(* IEC 61131-3 sources: elnaProjects/ElpcLogic/PomarKc7Changed/build_USO_ecl, 1 file *)

(* ---- plc.st ---- *)
TYPE
  TYPE_PhaseAlgoritmAction : (_run, _reset);
  TYPE_DualStateImAction : (_on, _off);
  struct_SectionSwitch : STRUCT
    inCommand : WORD;
    status : DWORD;
    onStatus : BYTE;
    inOpcCommandsDisabled : BOOL;
    sdvig : BOOL;
    Ns : BOOL;
    CommandFault : BOOL;
    Accident : BOOL;
    Local : BOOL;
    Distance : BOOL;
    OpcCommandsDisabled : BOOL;
    lastCmdIsOn : BOOL;
    offKNA : BOOL;
    basketStatus : BYTE;
    ISVALIDREF_statOn : BOOL;
    ISVALIDREF_statOff : BOOL;
    ISVALIDREF_cmdOn : BOOL;
    ISVALIDREF_cmdOff : BOOL;
    ISVALIDREF_inBreakCmdOn : BOOL;
    ISVALIDREF_inBreakCmdOff : BOOL;
    BreakCmdOn : BOOL;
    BreakCmdOff : BOOL;
    ISVALIDREF_basketRolledIn : BOOL;
    ISVALIDREF_basketRolledOut : BOOL;
    ISVALIDREF_basketTest : BOOL;
    inCommand_Alg : WORD;
    inCommand_ARM : WORD;
    cmdOn : BOOL;
    cmdOff : BOOL;
    reliability : BOOL;
  END_STRUCT;
  struct_ReserveIM2 : STRUCT
    var1 : BOOL;
    var2 : BOOL;
  END_STRUCT;
  struct_DiProtection : STRUCT
    delay : TIME;
    inTag : BYTE;
    inRunOnStart : BOOL;
    inCanRun : BOOL;
    inOpcCommandsDisabled : BOOL;
    inCommand : WORD;
    inCommand_Alg : WORD;
    inCommand_ARM : WORD;
    Tag : BYTE;
    status : DWORD;
    CanRun : BOOL;
    OpcCommandsDisabled : BOOL;
    isRunning : BOOL;
    HasError : BOOL;
    isEnded : BOOL;
    Remont : BOOL;
    Check : BOOL;
    Signaling : BOOL;
    SignalingTP : BOOL;
    RunOnStart : BOOL;
  END_STRUCT;
  TYPE_ReliableBit : STRUCT
    value : BOOL;
    reliability : BOOL;
    _inversed : BOOL;
  END_STRUCT;
  struct_DI : STRUCT
    imit : BOOL;
    value : WORD;
    reliability : WORD;
    bits : ARRAY [0..15] OF TYPE_ReliableBit;
    blConnect : BOOL;
  END_STRUCT;
  struct_AiProtection : STRUCT
    controlLimit : BYTE;
    delay : TIME;
    inTag : BYTE;
    inRunOnStart : BOOL;
    inCanRun : BOOL;
    inOpcCommandsDisabled : BOOL;
    inCommand : WORD;
    inCommand_Alg : WORD;
    inCommand_ARM : WORD;
    Tag : BYTE;
    status : DWORD;
    CanRun : BOOL;
    OpcCommandsDisabled : BOOL;
    isRunning : BOOL;
    HasError : BOOL;
    isEnded : BOOL;
    Remont : BOOL;
    Check : BOOL;
    Signaling : BOOL;
    SignalingTP : BOOL;
    RunOnStart : BOOL;
  END_STRUCT;
  ProtectionsConfig : STRUCT
    Topornogo_podshipnika_EDT_1 : struct_AiProtection;
    Toy_podshipnika_EDT_2 : struct_AiProtection;
    Toy_podshipnika_kol_EDT_3 : struct_AiProtection;
    Toy_podshipnika_kol_EDT_4 : struct_AiProtection;
    To_podshipnika_shest_red_EDT_5 : struct_AiProtection;
    To_podshipnika_shest_red_EDT_6 : struct_AiProtection;
    To_podshipnika_N_EDT_7 : struct_AiProtection;
    To_podshipnika_svob_konca_EDT_8 : struct_AiProtection;
    Ty_podshipnika_rab_kol_EDT_9 : struct_AiProtection;
    Typornogo_podshipnika_nerab_kolodok_HT_10 : struct_AiProtection;
    Tgaza_na_vyhode_H : struct_AiProtection;
    Os_sdvig_nagnetatelja_plus : struct_AiProtection;
    Os_sdvig_nagnetatelja_minus : struct_AiProtection;
    Pgaza_na_vyhode_nagnetatelia_GPA_STOP : struct_AiProtection;
    Pgaza_na_vhode_nagnetatelia_GPA_STOP : struct_AiProtection;
    Pgaza_na_vyhode_nagnetatelia : struct_AiProtection;
    dPmaslo_gaz : struct_AiProtection;
    Pmaslo_sm_nizkoe : struct_AiProtection;
    Pmaslo_sm_vysokoe : struct_AiProtection;
    Vibro_skorost_OPED_T1 : struct_AiProtection;
    Vibro_skorost_OPED_T2 : struct_AiProtection;
    Vibro_skorost_OYP_kolesa_ED_T3 : struct_AiProtection;
    Vibro_skorost_OP_kolesa_RH_T4 : struct_AiProtection;
    Vibro_skorost_OP_shesterni_RED_T5 : struct_AiProtection;
    Vibro_skorost_OP_shesterni_RED_T6 : struct_AiProtection;
    dPmaslo_gaz_less100 : struct_DiProtection;
    Reg_vozb_off : struct_DiProtection;
    Fail_chastotnii_pusk : struct_DiProtection;
    Off_avar_vikluchatel : struct_DiProtection;
    AOKC_SHKC : struct_DiProtection;
    AO_PRU : struct_DiProtection;
    AO_ot_SHU : struct_DiProtection;
    mvOff : struct_DiProtection;
    Kran1_sdvig : struct_DiProtection;
    Kran2_sdvig : struct_DiProtection;
  END_STRUCT;
  struct_singleSignal : STRUCT
    reliability : BOOL;
    inverse : BOOL;
    DelayOn : TIME;
    DelayOff : TIME;
    Q : BOOL;
    status : DWORD;
    Disabled_Sig : BOOL;
  END_STRUCT;
  IM_singleSignals : STRUCT
    dP_maslo_gaz_Less100 : struct_singleSignal;
    dp_kran1_Less100 : struct_singleSignal;
    Razreshenie_zagruzki_dvig : struct_singleSignal;
    Vozbud_gotovnost : struct_singleSignal;
    Vozbud_neispr_tsepey_upr_AVR_pit : struct_singleSignal;
    Vozbud_neispravnost : struct_singleSignal;
    SHAVR1_v_rabote : struct_singleSignal;
    SHAVR2_v_rabote : struct_singleSignal;
    Avariinoe_otkluch_vikluchatelya : struct_singleSignal;
    Assinhronnii_hod_peregruzka : struct_singleSignal;
    SHU_v_GPA_vkluch : struct_singleSignal;
    SHP_v_GPA_vkluch : struct_singleSignal;
    QF1_on : struct_singleSignal;
    QF2_on : struct_singleSignal;
    QF23_on : struct_singleSignal;
    QF4_QF5_on : struct_singleSignal;
    QF6_QF7_on : struct_singleSignal;
    QF8_QF9_on : struct_singleSignal;
    QF10_QF11_on : struct_singleSignal;
    QF12_QF13_on : struct_singleSignal;
    QF14_QF15_on : struct_singleSignal;
    QF22_on : struct_singleSignal;
    NS_G1_G2 : struct_singleSignal;
    NS_G3_G4 : struct_singleSignal;
    NS_G15_G16 : struct_singleSignal;
    NS_G17 : struct_singleSignal;
    NS_G5_G6 : struct_singleSignal;
    NS_G7_G8 : struct_singleSignal;
    NS_G18_G19 : struct_singleSignal;
    NS_G10_G11 : struct_singleSignal;
    NS_G13_G14 : struct_singleSignal;
    Uroven_masla_akkum : struct_singleSignal;
    NKU1_GPA_on : struct_singleSignal;
    NKU2_GPA_on : struct_singleSignal;
    AO_KC_ot_SHKS : struct_singleSignal;
    AO_GPA_ot_SHU : struct_singleSignal;
    BEAO_srabotal : struct_singleSignal;
    Chastotny_pusk : struct_singleSignal;
    Neuspesh_chastotny_pusk : struct_singleSignal;
    Rezhim_ruchnogo_regulirovaniya : struct_singleSignal;
    Osnovnoy_regul_off : struct_singleSignal;
    Voltage_sekcii_norm : struct_singleSignal;
    Reactorny_pusk : struct_singleSignal;
    NO_GPA_ot_SHU : struct_singleSignal;
    AO_GPA_ot_PRU : struct_singleSignal;
    Nalichie_BP1 : struct_singleSignal;
    Nalichie_BP2 : struct_singleSignal;
    Nalichie_BP3 : struct_singleSignal;
    Nalichie_BP4 : struct_singleSignal;
    Nalichie_BP5 : struct_singleSignal;
    Nalichie_BP6 : struct_singleSignal;
    Nalichie_BP7_BP8 : struct_singleSignal;
    Nalichie_BP9_BP10 : struct_singleSignal;
    Nalichie_cepei_upravlen_mv : struct_singleSignal;
    Nalichie_220BEAO : struct_singleSignal;
    Nalichie_per_220_na_vhode : struct_singleSignal;
    Nalichie_post_220_na_vhode : struct_singleSignal;
    Nalichie_BP11 : struct_singleSignal;
    Nalichie_BP12 : struct_singleSignal;
    Dver_SHU_pered_otkrita : struct_singleSignal;
    Dver_SHU_zad_otkrita : struct_singleSignal;
    EO_GPA_ot_knopki_SHU : struct_singleSignal;
    EO_EGPA_ot_PRY : struct_singleSignal;
    Synchroniz_rezhima_K1 : struct_singleSignal;
    Potok_ms_posle_AVOM : struct_singleSignal;
  END_STRUCT;
  DiConfig : STRUCT
    di_0 : struct_DI;
    di_1 : struct_DI;
    di_2 : struct_DI;
    di_3 : struct_DI;
    di_4 : struct_DI;
    di_5 : struct_DI;
    di_6 : struct_DI;
    di_7 : struct_DI;
    di_8 : struct_DI;
    di_9 : struct_DI;
    di_10 : struct_DI;
    di_11 : struct_DI;
    di_12 : struct_DI;
    di_13 : struct_DI;
    di_14 : struct_DI;
    di_15 : struct_DI;
    di_16 : struct_DI;
    di_17 : struct_DI;
    di_18 : struct_DI;
    di_19 : struct_DI;
    di_20 : struct_DI;
    di_21 : struct_DI;
  END_STRUCT;
  struct_AO : STRUCT
    nValue : LREAL;
    blConnect : BOOL;
    outLL : LREAL;
    outHL : LREAL;
    newLL : LREAL;
    newHL : LREAL;
    newLL_ISVALIDREF : BOOL;
    newHL_ISVALIDREF : BOOL;
    inCommand : WORD;
    Value : LREAL;
    status : DWORD;
    LL : LREAL;
    HL : LREAL;
    OpcCommandsDisabled : BOOL;
  END_STRUCT;
  AOConfig : STRUCT
    Reserv_AO_1 : struct_AO;
    Reserv_AO_2 : struct_AO;
  END_STRUCT;
  struct_AI : STRUCT
    value : LREAL;
    status : DWORD;
    interval : BYTE;
    inCommand : WORD;
    blConnect : BOOL;
    dLL : LREAL;
    dHL : LREAL;
    dLA : LREAL;
    dHA : LREAL;
    dLW : LREAL;
    dHW : LREAL;
    LL : LREAL;
    HL : LREAL;
    LA : LREAL;
    HA : LREAL;
    LW : LREAL;
    HW : LREAL;
    ISVALIDREF_LA : BOOL;
    ISVALIDREF_HA : BOOL;
    ISVALIDREF_LW : BOOL;
    ISVALIDREF_HW : BOOL;
    inpLL : LREAL;
    inpHL : LREAL;
    CurrentShotCircuit : LREAL;
    CurrentBreakCircuit : LREAL;
    maxChangeSpeed : LREAL;
    maxChangeSpeedDown : LREAL;
    ChangeSpeed : LREAL;
    histeresis : LREAL;
    aperturFilter : LREAL;
    exponentialFilter : LREAL;
    rassoglasovanie : LREAL;
    OpcCommandsDisabled : BOOL;
    Disabled_LA : BOOL;
    Disabled_HA : BOOL;
    Disabled_LW : BOOL;
    Disabled_HW : BOOL;
    delayLA : TIME;
    delayLW : TIME;
    delayHW : TIME;
    delayHA : TIME;
    minValue_ISVALIDREF : BOOL;
    maxValue_ISVALIDREF : BOOL;
    minValue : LREAL;
    maxValue : LREAL;
    inOpcCommandsDisabled : BOOL;
    imit : BOOL;
    remont : BOOL;
    NS : BOOL;
    NS_Min : BOOL;
    NS_Max : BOOL;
    inCommand_Alg : WORD;
    inCommand_ARM : WORD;
    dMaxChangeSpeed : LREAL;
    dMaxChangeSpeedDown : LREAL;
  END_STRUCT;
  AiConfig : STRUCT
    Tstali_statora_kanal_1 : struct_AI;
    Tstali_statora_kanal_2 : struct_AI;
    Tstali_statora_kanal_3 : struct_AI;
    Tmedi_statora_kanal_1 : struct_AI;
    Tmedi_statora_kanal_2 : struct_AI;
    Tmedi_statora_kanal_3 : struct_AI;
    Toporno_podshipnika_EDT_1 : struct_AI;
    Toy_podshipnika_EDT_2 : struct_AI;
    Toy_podshipnika_kol_EDT_3 : struct_AI;
    Toy_podshipnika_kol_EDT_4 : struct_AI;
    Toy_podshipnika_shest_red_EDT_5 : struct_AI;
    Ty_podshipnika_red_EDT_6 : struct_AI;
    Ty_podshipnika_nagnet_EDT_7_1 : struct_AI;
    Ty_podshipnika_nagnet_EDT_7_2 : struct_AI;
    Toy_podshipnika_svobod_konca_EDT_8_1 : struct_AI;
    Toy_podshipnika_svobod_konca_EDT_8_2 : struct_AI;
    Toy_podshipnika_rab_kol_EDT_9_1 : struct_AI;
    Toy_podshipnika_rab_kol_EDT_9_2 : struct_AI;
    Toy_podshipnika_nerab_kol_EDT_10_1 : struct_AI;
    Toy_podshipnika_nerab_kol_EDT_10_2 : struct_AI;
    Tholodnogo_vozduha_ED_kanal_1 : struct_AI;
    Tholodnogo_vozduha_ED_kanal_2 : struct_AI;
    Tgorjachego_vozduha_ED_kanal_1 : struct_AI;
    Tgorjachego_vozduha_ED_kanal_2 : struct_AI;
    Tnarujnogo_vozduha : struct_AI;
    Tgaza_na_vhode_H : struct_AI;
    Tgaza_na_vyhode_H : struct_AI;
    Tmasla_do_AVOM : struct_AI;
    Tmasla_posle_AVOM : struct_AI;
    Tmasla_MB : struct_AI;
    Tmasla_MB_TEN : struct_AI;
    Tshu : struct_AI;
    Pmaslo_sm_nizkoe : struct_AI;
    Pmaslo_sm_vysokoe : struct_AI;
    Pmasla_posle_GNS : struct_AI;
    Pmasla_posle_NU : struct_AI;
    Pgaza_na_vhode_nagnetatelia : struct_AI;
    Pgaza_na_vyhode_nagnetatelia : struct_AI;
    Pimpuls_gaz : struct_AI;
    dPgaza_na_maslo_filtre : struct_AI;
    dPgaza_na_konfuzore : struct_AI;
    dPmaslo_gaz : struct_AI;
    Os_sdvig_nagnetatelja_plus : struct_AI;
    Os_sdvig_nagnetatelja_minus : struct_AI;
    Yroven_masla_MB : struct_AI;
    Kontrol_per_220V : struct_AI;
    Kontrol_post_220V : struct_AI;
    Tok_statora : struct_AI;
    Vibro_skorost_OPED_T1 : struct_AI;
    Vibro_skorost_OYPED_T2 : struct_AI;
    Vibro_skorost_OYP_kolesa_ED_T3 : struct_AI;
    Vibro_skorost_OP_kolesa_RH_T4 : struct_AI;
    Vibro_skorost_OP_shesterni_RED_T5 : struct_AI;
    Vibro_skorost_OP_shesterni_RED_T6 : struct_AI;
  END_STRUCT;
  TYPE_ProtectionTags : STRUCT
    NOTHING : BYTE := 0;
    AOB : BYTE := 1;
    AOS : BYTE := 2;
    AOPOJ : BYTE := 3;
  END_STRUCT;
  TYPE_ModeGpa : STRUCT
    MODE_NOTDEFINED : UINT := 0;
    MODE_REMONT : UINT := 1;
    MODE_STOP : UINT := 2;
    MODE_READY : UINT := 3;
    MODE_PUSKV : UINT := 4;
    MODE_PUSKK : UINT := 5;
    MODE_TESTDPMG : UINT := 6;
    MODE_TESTPMS : UINT := 7;
    MODE_APUSK : UINT := 8;
    MODE_MPUSK : UINT := 9;
    MODE_WORK_Ring : UINT := 10;
    MODE_WORK_Line : UINT := 11;
    MODE_NO : UINT := 12;
    MODE_AO : UINT := 13;
    MODE_EO : UINT := 14;
    MODE_TESTIM : UINT := 15;
    MODE_TESTAZ : UINT := 16;
    MODE_PUSK_FIRST_FAZA1 : UINT := 17;
    MODE_PUSK_FIRST_FAZA2 : UINT := 18;
  END_STRUCT;
  struct_DualStateIm : STRUCT
    inCommand : WORD;
    status : DWORD;
    onStatus : BYTE;
    inOpcCommandsDisabled : BOOL;
    sdvig : BOOL;
    Ns : BOOL;
    CommandFault : BOOL;
    Accident : BOOL;
    OpcCommandsDisabled : BOOL;
    lastCmdIsOn : BOOL;
    ISVALIDREF_statOn : BOOL;
    ISVALIDREF_statOff : BOOL;
    ISVALIDREF_cmdOn : BOOL;
    ISVALIDREF_cmdOff : BOOL;
    inCommand_Alg : WORD;
    inCommand_ARM : WORD;
    cmdOn : BOOL;
    cmdOff : BOOL;
    reliability : BOOL;
  END_STRUCT;
  struct_DO : STRUCT
    imit : BOOL;
    blConnect : BOOL;
    value : WORD;
    bits : ARRAY [0..15] OF BOOL;
  END_STRUCT;
  struct_AlgTimers : STRUCT
    AutoPns_OffTimer : UINT;
    AutoPns_OnTimer : UINT;
    vibegPNS_Timer : UINT;
    NO_waitCloseKran : UINT;
    AO_waitKran : UINT;
    testPms_BreakTest : UINT;
    testdPmg_BreakTest : UINT;
    puskOilSystem_BreakPuskTimer_Poil : UINT;
    engineRun_BreakPuskTimer : UINT;
    filling_BreakPuskTimer : UINT;
    filling_waitAfterKran4 : UINT;
    filling_waitAfterKran5 : UINT;
    puskK_wait720 : UINT;
    puskV_wait600 : UINT;
    No_wait120 : UINT;
    No_wait600 : UINT;
    No_wait5 : UINT;
  END_STRUCT;
  struct_AlgoritmsManager : STRUCT
    mode : UINT;
    narabotka : UINT;
    nMode : UINT;
    AnalogsPs : BOOL;
    DiscretPS : BOOL;
    ProtectionSignaling : BOOL;
  END_STRUCT;
  struct_Alg : STRUCT
    inRunOnStart : BOOL;
    inCanRun : BOOL;
    inHasError : BOOL;
    inEnded : BOOL;
    inOpcCommandsDisabled : BOOL;
    inCommand : WORD;
    inCommand_ARM : WORD;
    inCommand_Alg : WORD;
    status : DWORD;
    CanRun : BOOL;
    OpcCommandsDisabled : BOOL;
    isRuning : BOOL;
    HasError : BOOL;
    isEnded : BOOL;
    RunOnStart : BOOL;
    Start : DWORD;
    Error : DWORD;
    Top : DWORD;
  END_STRUCT;
  struct_singleOutput : STRUCT
    wait_time : TIME;
    inCommand : WORD;
    inOpcCommandsDisabled : BOOL;
    Q : BOOL;
    status : DWORD;
    OpcCommandsDisabled : BOOL;
    inCommand_Alg : WORD;
    inCommand_ARM : WORD;
  END_STRUCT;
  IM_singleOutputs : STRUCT
    Rabota_EGPA : struct_singleOutput;
    Neispr_EGPA : struct_singleOutput;
    Avary_EGPA : struct_singleOutput;
    U_lamp_SHU : struct_singleOutput;
    AO_knopka_ind : struct_singleOutput;
    Pusk_SHUP : struct_singleOutput;
    Stop_SHUP : struct_singleOutput;
    NO_fonar : struct_singleOutput;
    PC_fonar : struct_singleOutput;
    AC_fonar : struct_singleOutput;
    Kr1_smazka : struct_singleOutput;
    Kr2_smazka : struct_singleOutput;
    Kr4_open_from_alg : struct_singleOutput;
    Synch_rej_K1 : struct_singleOutput;
  END_STRUCT;
  DOconfig : STRUCT
    do_0 : struct_DO;
    do_1 : struct_DO;
    do_2 : struct_DO;
    do_3 : struct_DO;
    do_4 : struct_DO;
    gpio_out : struct_DO;
  END_STRUCT;
  struct_Question : STRUCT
    AnswerVariants : UINT;
    inCommand : WORD;
    ask : BOOL;
    reset : BOOL;
    status : DWORD;
    answer : UINT;
    OpcCommandsDisabled : BOOL;
    inOpcCommandsDisabled : BOOL;
  END_STRUCT;
  AlgoritmsQuestions : STRUCT
    vibegPNS_algContinue : struct_Question;
    testPms_algContinue : struct_Question;
    testdPmg_algContinue : struct_Question;
    puskK_questionFilling : struct_Question;
    puskK_questionUnload : struct_Question;
    puskV_questionEngine : struct_Question;
    puskV_questionMVoff : struct_Question;
    SemiAutoPusk_cmdRun1ph : struct_Question;
    SemiAutoPusk_cmdRun2ph : struct_Question;
    SemiAutoPusk_cmdRun3ph : struct_Question;
    SemiAutoPusk_cmdRun4ph : struct_Question;
  END_STRUCT;
  TYPE_Answers : STRUCT
    ANS_NONE : UINT := 0;
    ANS_YES : UINT := 1;
    ANS_NO : UINT := 2;
    ANS_CANCEL : UINT := 4;
    ANS_RETRY : UINT := 8;
  END_STRUCT;
  TYPE_AnalogLimitFlags : STRUCT
    NONE : BYTE := 0;
    LL : BYTE := 16#1;
    LW : BYTE := 16#2;
    HW : BYTE := 16#4;
    LA : BYTE := 16#8;
    HA : BYTE := 16#10;
    HL : BYTE := 16#20;
    SipUP : BYTE := 16#40;
    SipDown : BYTE := 16#80;
  END_STRUCT;
  struct_AnalogParametr : STRUCT
    inCommand : WORD;
    inCommand_Alg : WORD;
    inCommand_ARM : WORD;
    status : DWORD;
    newValue : LREAL;
    currentValue : LREAL;
    minVal : LREAL;
    maxVal : LREAL;
    maxStep : LREAL;
    minVal_ISVALIDREF : BOOL;
    maxVal_ISVALIDREF : BOOL;
    maxStep_ISVALIDREF : BOOL;
    inOpcCommandsDisabled : BOOL;
    Value : LREAL;
    isValidValue : BOOL;
    OpcCommandsDisabled : BOOL;
  END_STRUCT;
  struct_Kran : STRUCT
    inCommand : WORD;
    status : DWORD;
    onStatus : BYTE;
    inOpcCommandsDisabled : BOOL;
    sdvig : BOOL;
    Ns : BOOL;
    Dp : BOOL;
    CommandFault : BOOL;
    Accident : BOOL;
    Auto : BOOL;
    Manual : BOOL;
    Local : BOOL;
    Distance : BOOL;
    ErrorPowerOff : BOOL;
    ErrorBlock : BOOL;
    So : BOOL;
    Sz : BOOL;
    OpcCommandsDisabled : BOOL;
    lastCmdIsOn : BOOL;
    ISVALIDREF_statOn : BOOL;
    ISVALIDREF_statOff : BOOL;
    ISVALIDREF_cmdOn : BOOL;
    ISVALIDREF_cmdOff : BOOL;
    ISVALIDREF_inSo : BOOL;
    ISVALIDREF_inSz : BOOL;
    ISVALIDREF_inDp : BOOL;
    continueHoldCommand : TIME;
    inCommand_Alg : WORD;
    inCommand_ARM : WORD;
    cmdOn : BOOL;
    cmdOff : BOOL;
    reliability : BOOL;
  END_STRUCT;
  struct_OilPump : STRUCT
    inCommand : WORD;
    inCommand_Alg : WORD;
    inCommand_ARM : WORD;
    status : DWORD;
    onStatus : BYTE;
    inOpcCommandsDisabled : BOOL;
    sdvig : BOOL;
    Ns : BOOL;
    CommandFault : BOOL;
    Accident : BOOL;
    Local : BOOL;
    Distance : BOOL;
    BreakCmdOn : BOOL;
    BreakCmdOff : BOOL;
    OpcCommandsDisabled : BOOL;
    lastCmdIsOn : BOOL;
    ISVALIDREF_statOn : BOOL;
    ISVALIDREF_statOff : BOOL;
    ISVALIDREF_cmdOn : BOOL;
    ISVALIDREF_cmdOff : BOOL;
    ISVALIDREF_inBreakCmdOn : BOOL;
    ISVALIDREF_inBreakCmdOff : BOOL;
    inBlocked : BOOL;
    Blocked : BOOL;
    Osnovnoy : BOOL;
    Rezervny : BOOL;
    cmdOn : BOOL;
    cmdOff : BOOL;
    reliability : BOOL;
  END_STRUCT;
  struct_Switch : STRUCT
    inCommand : WORD;
    status : DWORD;
    onStatus : BYTE;
    inOpcCommandsDisabled : BOOL;
    sdvig : BOOL;
    Ns : BOOL;
    CommandFault : BOOL;
    Accident : BOOL;
    Auto : BOOL;
    Manual : BOOL;
    Local : BOOL;
    Distance : BOOL;
    ErrorPowerOff : BOOL;
    ErrorBlock : BOOL;
    BreakCmdOn : BOOL;
    BreakCmdOff : BOOL;
    OpcCommandsDisabled : BOOL;
    lastCmdIsOn : BOOL;
    ISVALIDREF_statOn : BOOL;
    ISVALIDREF_statOff : BOOL;
    ISVALIDREF_cmdOn : BOOL;
    ISVALIDREF_cmdOff : BOOL;
    ISVALIDREF_inBreakCmdOn : BOOL;
    ISVALIDREF_inBreakCmdOff : BOOL;
    inCommand_Alg : WORD;
    inCommand_ARM : WORD;
    cmdOn : BOOL;
    cmdOff : BOOL;
    reliability : BOOL;
  END_STRUCT;
  struct_ReserveIM : STRUCT
    var1 : BOOL;
    var2 : BOOL;
  END_STRUCT;
  ImConfig : STRUCT
    Kran1 : struct_Kran;
    Kran2 : struct_Kran;
    Kran3 : struct_Kran;
    Kran3b : struct_Kran;
    Kran4 : struct_Kran;
    Kran5 : struct_Kran;
    Kran6 : struct_Kran;
    nu1 : struct_OilPump;
    nu2 : struct_OilPump;
    pns : struct_Switch;
    v1_Avom : struct_Switch;
    v2_Avom : struct_Switch;
    v3_Avom : struct_Switch;
    v4_Avom : struct_Switch;
    mv : struct_SectionSwitch;
    Reserve_IM1 : struct_ReserveIM;
    Reserve_IM2 : struct_ReserveIM2;
    SingleSignals : IM_singleSignals;
    SingleOutputs : IM_singleOutputs;
    KaloriferAVOM : struct_Switch;
    CMN : struct_Switch;
    TEN_kollectora : struct_Switch;
    TEN_MB : struct_Switch;
  END_STRUCT;
  AlgoritmsConfig : STRUCT
    autoNu : struct_Alg;
    AutoPns : struct_Alg;
    AutoAvom : struct_Alg;
    AutoTen : struct_Alg;
    AntiPompag : struct_Alg;
    testIm : struct_Alg;
    TestProtection : struct_Alg;
    Remont : struct_Alg;
    ppu : struct_Alg;
    puskOilSystem : struct_Alg;
    engineRun : struct_Alg;
    filling : struct_Alg;
    LineToRing : struct_Alg;
    RingToLine : struct_Alg;
    Apusk : struct_Alg;
    SemiAutoPusk : struct_Alg;
    no : struct_Alg;
    vibegPNS : struct_Alg;
    ao : struct_Alg;
    testPms : struct_Alg;
    testdPmg : struct_Alg;
    puskV : struct_Alg;
    puskK : struct_Alg;
    Pusk_F_faza1 : struct_Alg;
    Pusk_F_faza2 : struct_Alg;
    Pusk_TH_faza : struct_Alg;
    Prov_PMS_ALG : struct_Alg;
    Prov_opressovka_ALG : struct_Alg;
    Pusk_SEC_faza_chastotny : struct_Alg;
    Pusk_SEC_faza_reactor : struct_Alg;
  END_STRUCT;
  TYPE_basketStats : STRUCT
    BASKET_NOTDEFINED : BYTE := 0;
    BASKET_ROLLEDIN : BYTE := 1;
    BASKET_ROLLEDOUT : BYTE := 2;
    BASKET_TRANSITIONAL : BYTE := 3;
    BASKET_ERROR : BYTE := 4;
    BASKET_TEST : BYTE := 5;
  END_STRUCT;
  struct_ProtectionsManager : STRUCT
    inCommand : BYTE;
    protectionInRemont : BOOL;
  END_STRUCT;
  struct_DiscretParametr : STRUCT
    newValue : UINT;
    currentValue : UINT;
    inOpcCommandsDisabled : BOOL;
    inCommand : WORD;
    inCommand_Alg : WORD;
    inCommand_ARM : WORD;
    status : DWORD;
    OpcCommandsDisabled : BOOL;
    Value : UINT;
  END_STRUCT;
  TYPE_TableRec : STRUCT
    x : REAL;
    y : REAL;
  END_STRUCT;
  TItemAIN : STRUCT
    wFlags : UINT := 0;
    wReserved : UINT := 0;
    dblValue : LREAL := 0.0;
    nanosec : ULINT := 0;
    reserve : ULINT := 0;
  END_STRUCT;
  TWordData : STRUCT
    wFlags : UINT := 0;
    wValue : UINT := 0;
  END_STRUCT;
  struct_PhaseAlgoritm : STRUCT
    run : BOOL;
    reset : BOOL;
    start : BOOL;
    error : BOOL;
    top : BOOL;
    startStatus : DWORD;
    errorStatus : DWORD;
    topStatus : DWORD;
  END_STRUCT;
  TYPE_commandDualInput : STRUCT
    CMD_ON : BYTE := 1;
    CMD_OFF : BYTE := 2;
    CMD_RESET : BYTE := 3;
  END_STRUCT;
  TYPE_StatusAi : STRUCT
    NOTDEFINED : BYTE := 0;
    LL : BYTE := 1;
    HL : BYTE := 2;
    NOTRELIABLE : BYTE := 3;
    normal : BYTE := 4;
    LW : BYTE := 5;
    HW : BYTE := 6;
    LA : BYTE := 7;
    HA : BYTE := 8;
  END_STRUCT;
  TItemDIN : STRUCT
    wFlags : UINT := 0;
    wValue : UINT := 0;
    nanosec : ULINT := 0;
    reserve : ULINT := 0;
  END_STRUCT;
  TYPE_statusDualInput : STRUCT
    STATUS_NOTDEFINED : BYTE := 0;
    STATUS_ON : BYTE := 1;
    STATUS_OFF : BYTE := 2;
    STATUS_TRANSITIONAL : BYTE := 3;
    STATUS_ERROR : BYTE := 4;
  END_STRUCT;
  TDoubleData : STRUCT
    wFlags : UINT := 0;
    dblValue : LREAL := 0.0;
  END_STRUCT;
  TYPE_CommandAnalog : STRUCT
    cmd_SetUstavki : WORD := 1;
    cmd_SetRemont : WORD := 2;
    cmd_ResetRemont : WORD := 3;
    cmd_kvitNotReliable : WORD := 4;
  END_STRUCT;
  TYPE_CommandsPotectionsManager : STRUCT
    RestartAllSignaling : BYTE := 1;
    RestartAllProtections : BYTE := 2;
    CheckProtections : BYTE := 3;
    ResetAllProtections : BYTE := 4;
  END_STRUCT;
END_TYPE

FUNCTION_BLOCK OPC_AI_INIT
  VAR_EXTERNAL
    ai : aiConfig;
    AI_Tstali_statora_kanal_1_HL : LREAL;
    AI_Tstali_statora_kanal_1_LL : LREAL;
    AI_Tstali_statora_kanal_1_command : UINT;
    AI_Tstali_statora_kanal_1_newHL : LREAL;
    AI_Tstali_statora_kanal_1_newLL : LREAL;
    AI_Tstali_statora_kanal_1_status : UDINT;
    AI_Tstali_statora_kanal_1_value : LREAL;
    AI_Tstali_statora_kanal_1_HW : LREAL;
    AI_Tstali_statora_kanal_1_newHW : LREAL;
    AI_Tstali_statora_kanal_2_HL : LREAL;
    AI_Tstali_statora_kanal_2_LL : LREAL;
    AI_Tstali_statora_kanal_2_command : UINT;
    AI_Tstali_statora_kanal_2_newHL : LREAL;
    AI_Tstali_statora_kanal_2_newLL : LREAL;
    AI_Tstali_statora_kanal_2_status : UDINT;
    AI_Tstali_statora_kanal_2_value : LREAL;
    AI_Tstali_statora_kanal_2_HW : LREAL;
    AI_Tstali_statora_kanal_2_newHW : LREAL;
    AI_Tstali_statora_kanal_3_HL : LREAL;
    AI_Tstali_statora_kanal_3_LL : LREAL;
    AI_Tstali_statora_kanal_3_command : UINT;
    AI_Tstali_statora_kanal_3_newHL : LREAL;
    AI_Tstali_statora_kanal_3_newLL : LREAL;
    AI_Tstali_statora_kanal_3_status : UDINT;
    AI_Tstali_statora_kanal_3_value : LREAL;
    AI_Tstali_statora_kanal_3_HW : LREAL;
    AI_Tstali_statora_kanal_3_newHW : LREAL;
    AI_Tmedi_statora_kanal_1_HL : LREAL;
    AI_Tmedi_statora_kanal_1_LL : LREAL;
    AI_Tmedi_statora_kanal_1_command : UINT;
    AI_Tmedi_statora_kanal_1_newHL : LREAL;
    AI_Tmedi_statora_kanal_1_newLL : LREAL;
    AI_Tmedi_statora_kanal_1_status : UDINT;
    AI_Tmedi_statora_kanal_1_value : LREAL;
    AI_Tmedi_statora_kanal_1_HW : LREAL;
    AI_Tmedi_statora_kanal_1_newHW : LREAL;
    AI_Tmedi_statora_kanal_2_HL : LREAL;
    AI_Tmedi_statora_kanal_2_LL : LREAL;
    AI_Tmedi_statora_kanal_2_command : UINT;
    AI_Tmedi_statora_kanal_2_newHL : LREAL;
    AI_Tmedi_statora_kanal_2_newLL : LREAL;
    AI_Tmedi_statora_kanal_2_status : UDINT;
    AI_Tmedi_statora_kanal_2_value : LREAL;
    AI_Tmedi_statora_kanal_2_HW : LREAL;
    AI_Tmedi_statora_kanal_2_newHW : LREAL;
    AI_Tmedi_statora_kanal_3_HL : LREAL;
    AI_Tmedi_statora_kanal_3_LL : LREAL;
    AI_Tmedi_statora_kanal_3_command : UINT;
    AI_Tmedi_statora_kanal_3_newHL : LREAL;
    AI_Tmedi_statora_kanal_3_newLL : LREAL;
    AI_Tmedi_statora_kanal_3_status : UDINT;
    AI_Tmedi_statora_kanal_3_value : LREAL;
    AI_Tmedi_statora_kanal_3_HW : LREAL;
    AI_Tmedi_statora_kanal_3_newHW : LREAL;
    AI_Toporno_podshipnika_EDT_1_HL : LREAL;
    AI_Toporno_podshipnika_EDT_1_LL : LREAL;
    AI_Toporno_podshipnika_EDT_1_command : UINT;
    AI_Toporno_podshipnika_EDT_1_newHL : LREAL;
    AI_Toporno_podshipnika_EDT_1_newLL : LREAL;
    AI_Toporno_podshipnika_EDT_1_status : UDINT;
    AI_Toporno_podshipnika_EDT_1_value : LREAL;
    AI_Toporno_podshipnika_EDT_1_HW : LREAL;
    AI_Toporno_podshipnika_EDT_1_newHW : LREAL;
    AI_Toporno_podshipnika_EDT_1_HA : LREAL;
    AI_Toporno_podshipnika_EDT_1_newHA : LREAL;
    AI_Toy_podshipnika_EDT_2_HL : LREAL;
    AI_Toy_podshipnika_EDT_2_LL : LREAL;
    AI_Toy_podshipnika_EDT_2_command : UINT;
    AI_Toy_podshipnika_EDT_2_newHL : LREAL;
    AI_Toy_podshipnika_EDT_2_newLL : LREAL;
    AI_Toy_podshipnika_EDT_2_status : UDINT;
    AI_Toy_podshipnika_EDT_2_value : LREAL;
    AI_Toy_podshipnika_EDT_2_HW : LREAL;
    AI_Toy_podshipnika_EDT_2_newHW : LREAL;
    AI_Toy_podshipnika_EDT_2_HA : LREAL;
    AI_Toy_podshipnika_EDT_2_newHA : LREAL;
    AI_Toy_podshipnika_kol_EDT_3_HL : LREAL;
    AI_Toy_podshipnika_kol_EDT_3_LL : LREAL;
    AI_Toy_podshipnika_kol_EDT_3_command : UINT;
    AI_Toy_podshipnika_kol_EDT_3_newHL : LREAL;
    AI_Toy_podshipnika_kol_EDT_3_newLL : LREAL;
    AI_Toy_podshipnika_kol_EDT_3_status : UDINT;
    AI_Toy_podshipnika_kol_EDT_3_value : LREAL;
    AI_Toy_podshipnika_kol_EDT_3_HW : LREAL;
    AI_Toy_podshipnika_kol_EDT_3_newHW : LREAL;
    AI_Toy_podshipnika_kol_EDT_3_HA : LREAL;
    AI_Toy_podshipnika_kol_EDT_3_newHA : LREAL;
    AI_Toy_podshipnika_kol_EDT_4_HL : LREAL;
    AI_Toy_podshipnika_kol_EDT_4_LL : LREAL;
    AI_Toy_podshipnika_kol_EDT_4_command : UINT;
    AI_Toy_podshipnika_kol_EDT_4_newHL : LREAL;
    AI_Toy_podshipnika_kol_EDT_4_newLL : LREAL;
    AI_Toy_podshipnika_kol_EDT_4_status : UDINT;
    AI_Toy_podshipnika_kol_EDT_4_value : LREAL;
    AI_Toy_podshipnika_kol_EDT_4_HW : LREAL;
    AI_Toy_podshipnika_kol_EDT_4_newHW : LREAL;
    AI_Toy_podshipnika_kol_EDT_4_HA : LREAL;
    AI_Toy_podshipnika_kol_EDT_4_newHA : LREAL;
    AI_Toy_podshipnika_shest_red_EDT_5_HL : LREAL;
    AI_Toy_podshipnika_shest_red_EDT_5_LL : LREAL;
    AI_Toy_podshipnika_shest_red_EDT_5_command : UINT;
    AI_Toy_podshipnika_shest_red_EDT_5_newHL : LREAL;
    AI_Toy_podshipnika_shest_red_EDT_5_newLL : LREAL;
    AI_Toy_podshipnika_shest_red_EDT_5_status : UDINT;
    AI_Toy_podshipnika_shest_red_EDT_5_value : LREAL;
    AI_Toy_podshipnika_shest_red_EDT_5_HW : LREAL;
    AI_Toy_podshipnika_shest_red_EDT_5_newHW : LREAL;
    AI_Toy_podshipnika_shest_red_EDT_5_HA : LREAL;
    AI_Toy_podshipnika_shest_red_EDT_5_newHA : LREAL;
    AI_Ty_podshipnika_red_EDT_6_HL : LREAL;
    AI_Ty_podshipnika_red_EDT_6_LL : LREAL;
    AI_Ty_podshipnika_red_EDT_6_command : UINT;
    AI_Ty_podshipnika_red_EDT_6_newHL : LREAL;
    AI_Ty_podshipnika_red_EDT_6_newLL : LREAL;
    AI_Ty_podshipnika_red_EDT_6_status : UDINT;
    AI_Ty_podshipnika_red_EDT_6_value : LREAL;
    AI_Ty_podshipnika_red_EDT_6_HW : LREAL;
    AI_Ty_podshipnika_red_EDT_6_newHW : LREAL;
    AI_Ty_podshipnika_red_EDT_6_HA : LREAL;
    AI_Ty_podshipnika_red_EDT_6_newHA : LREAL;
    AI_Ty_podshipnika_nagnet_EDT_7_1_HL : LREAL;
    AI_Ty_podshipnika_nagnet_EDT_7_1_LL : LREAL;
    AI_Ty_podshipnika_nagnet_EDT_7_1_command : UINT;
    AI_Ty_podshipnika_nagnet_EDT_7_1_newHL : LREAL;
    AI_Ty_podshipnika_nagnet_EDT_7_1_newLL : LREAL;
    AI_Ty_podshipnika_nagnet_EDT_7_1_status : UDINT;
    AI_Ty_podshipnika_nagnet_EDT_7_1_value : LREAL;
    AI_Ty_podshipnika_nagnet_EDT_7_1_HW : LREAL;
    AI_Ty_podshipnika_nagnet_EDT_7_1_newHW : LREAL;
    AI_Ty_podshipnika_nagnet_EDT_7_1_HA : LREAL;
    AI_Ty_podshipnika_nagnet_EDT_7_1_newHA : LREAL;
    AI_Ty_podshipnika_nagnet_EDT_7_2_HL : LREAL;
    AI_Ty_podshipnika_nagnet_EDT_7_2_LL : LREAL;
    AI_Ty_podshipnika_nagnet_EDT_7_2_command : UINT;
    AI_Ty_podshipnika_nagnet_EDT_7_2_newHL : LREAL;
    AI_Ty_podshipnika_nagnet_EDT_7_2_newLL : LREAL;
    AI_Ty_podshipnika_nagnet_EDT_7_2_status : UDINT;
    AI_Ty_podshipnika_nagnet_EDT_7_2_value : LREAL;
    AI_Ty_podshipnika_nagnet_EDT_7_2_HW : LREAL;
    AI_Ty_podshipnika_nagnet_EDT_7_2_newHW : LREAL;
    AI_Ty_podshipnika_nagnet_EDT_7_2_HA : LREAL;
    AI_Ty_podshipnika_nagnet_EDT_7_2_newHA : LREAL;
    AI_Toy_podshipnika_svobod_konca_EDT_8_1_HL : LREAL;
    AI_Toy_podshipnika_svobod_konca_EDT_8_1_LL : LREAL;
    AI_Toy_podshipnika_svobod_konca_EDT_8_1_command : UINT;
    AI_Toy_podshipnika_svobod_konca_EDT_8_1_newHL : LREAL;
    AI_Toy_podshipnika_svobod_konca_EDT_8_1_newLL : LREAL;
    AI_Toy_podshipnika_svobod_konca_EDT_8_1_status : UDINT;
    AI_Toy_podshipnika_svobod_konca_EDT_8_1_value : LREAL;
    AI_Toy_podshipnika_svobod_konca_EDT_8_1_HW : LREAL;
    AI_Toy_podshipnika_svobod_konca_EDT_8_1_newHW : LREAL;
    AI_Toy_podshipnika_svobod_konca_EDT_8_1_HA : LREAL;
    AI_Toy_podshipnika_svobod_konca_EDT_8_1_newHA : LREAL;
    AI_Toy_podshipnika_svobod_konca_EDT_8_2_HL : LREAL;
    AI_Toy_podshipnika_svobod_konca_EDT_8_2_LL : LREAL;
    AI_Toy_podshipnika_svobod_konca_EDT_8_2_command : UINT;
    AI_Toy_podshipnika_svobod_konca_EDT_8_2_newHL : LREAL;
    AI_Toy_podshipnika_svobod_konca_EDT_8_2_newLL : LREAL;
    AI_Toy_podshipnika_svobod_konca_EDT_8_2_status : UDINT;
    AI_Toy_podshipnika_svobod_konca_EDT_8_2_value : LREAL;
    AI_Toy_podshipnika_svobod_konca_EDT_8_2_HW : LREAL;
    AI_Toy_podshipnika_svobod_konca_EDT_8_2_newHW : LREAL;
    AI_Toy_podshipnika_svobod_konca_EDT_8_2_HA : LREAL;
    AI_Toy_podshipnika_svobod_konca_EDT_8_2_newHA : LREAL;
    AI_Toy_podshipnika_rab_kol_EDT_9_1_HL : LREAL;
    AI_Toy_podshipnika_rab_kol_EDT_9_1_LL : LREAL;
    AI_Toy_podshipnika_rab_kol_EDT_9_1_command : UINT;
    AI_Toy_podshipnika_rab_kol_EDT_9_1_newHL : LREAL;
    AI_Toy_podshipnika_rab_kol_EDT_9_1_newLL : LREAL;
    AI_Toy_podshipnika_rab_kol_EDT_9_1_status : UDINT;
    AI_Toy_podshipnika_rab_kol_EDT_9_1_value : LREAL;
    AI_Toy_podshipnika_rab_kol_EDT_9_1_HW : LREAL;
    AI_Toy_podshipnika_rab_kol_EDT_9_1_newHW : LREAL;
    AI_Toy_podshipnika_rab_kol_EDT_9_1_HA : LREAL;
    AI_Toy_podshipnika_rab_kol_EDT_9_1_newHA : LREAL;
    AI_Toy_podshipnika_rab_kol_EDT_9_2_HL : LREAL;
    AI_Toy_podshipnika_rab_kol_EDT_9_2_LL : LREAL;
    AI_Toy_podshipnika_rab_kol_EDT_9_2_command : UINT;
    AI_Toy_podshipnika_rab_kol_EDT_9_2_newHL : LREAL;
    AI_Toy_podshipnika_rab_kol_EDT_9_2_newLL : LREAL;
    AI_Toy_podshipnika_rab_kol_EDT_9_2_status : UDINT;
    AI_Toy_podshipnika_rab_kol_EDT_9_2_value : LREAL;
    AI_Toy_podshipnika_rab_kol_EDT_9_2_HW : LREAL;
    AI_Toy_podshipnika_rab_kol_EDT_9_2_newHW : LREAL;
    AI_Toy_podshipnika_rab_kol_EDT_9_2_HA : LREAL;
    AI_Toy_podshipnika_rab_kol_EDT_9_2_newHA : LREAL;
    AI_Toy_podshipnika_nerab_kol_EDT_10_1_HL : LREAL;
    AI_Toy_podshipnika_nerab_kol_EDT_10_1_LL : LREAL;
    AI_Toy_podshipnika_nerab_kol_EDT_10_1_command : UINT;
    AI_Toy_podshipnika_nerab_kol_EDT_10_1_newHL : LREAL;
    AI_Toy_podshipnika_nerab_kol_EDT_10_1_newLL : LREAL;
    AI_Toy_podshipnika_nerab_kol_EDT_10_1_status : UDINT;
    AI_Toy_podshipnika_nerab_kol_EDT_10_1_value : LREAL;
    AI_Toy_podshipnika_nerab_kol_EDT_10_1_HW : LREAL;
    AI_Toy_podshipnika_nerab_kol_EDT_10_1_newHW : LREAL;
    AI_Toy_podshipnika_nerab_kol_EDT_10_1_HA : LREAL;
    AI_Toy_podshipnika_nerab_kol_EDT_10_1_newHA : LREAL;
    AI_Toy_podshipnika_nerab_kol_EDT_10_2_HL : LREAL;
    AI_Toy_podshipnika_nerab_kol_EDT_10_2_LL : LREAL;
    AI_Toy_podshipnika_nerab_kol_EDT_10_2_command : UINT;
    AI_Toy_podshipnika_nerab_kol_EDT_10_2_newHL : LREAL;
    AI_Toy_podshipnika_nerab_kol_EDT_10_2_newLL : LREAL;
    AI_Toy_podshipnika_nerab_kol_EDT_10_2_status : UDINT;
    AI_Toy_podshipnika_nerab_kol_EDT_10_2_value : LREAL;
    AI_Toy_podshipnika_nerab_kol_EDT_10_2_HW : LREAL;
    AI_Toy_podshipnika_nerab_kol_EDT_10_2_newHW : LREAL;
    AI_Toy_podshipnika_nerab_kol_EDT_10_2_HA : LREAL;
    AI_Toy_podshipnika_nerab_kol_EDT_10_2_newHA : LREAL;
    AI_Tholodnogo_vozduha_ED_kanal_1_HL : LREAL;
    AI_Tholodnogo_vozduha_ED_kanal_1_LL : LREAL;
    AI_Tholodnogo_vozduha_ED_kanal_1_command : UINT;
    AI_Tholodnogo_vozduha_ED_kanal_1_newHL : LREAL;
    AI_Tholodnogo_vozduha_ED_kanal_1_newLL : LREAL;
    AI_Tholodnogo_vozduha_ED_kanal_1_status : UDINT;
    AI_Tholodnogo_vozduha_ED_kanal_1_value : LREAL;
    AI_Tholodnogo_vozduha_ED_kanal_1_HW : LREAL;
    AI_Tholodnogo_vozduha_ED_kanal_1_newHW : LREAL;
    AI_Tholodnogo_vozduha_ED_kanal_2_HL : LREAL;
    AI_Tholodnogo_vozduha_ED_kanal_2_LL : LREAL;
    AI_Tholodnogo_vozduha_ED_kanal_2_command : UINT;
    AI_Tholodnogo_vozduha_ED_kanal_2_newHL : LREAL;
    AI_Tholodnogo_vozduha_ED_kanal_2_newLL : LREAL;
    AI_Tholodnogo_vozduha_ED_kanal_2_status : UDINT;
    AI_Tholodnogo_vozduha_ED_kanal_2_value : LREAL;
    AI_Tholodnogo_vozduha_ED_kanal_2_HW : LREAL;
    AI_Tholodnogo_vozduha_ED_kanal_2_newHW : LREAL;
    AI_Tgorjachego_vozduha_ED_kanal_1_HL : LREAL;
    AI_Tgorjachego_vozduha_ED_kanal_1_LL : LREAL;
    AI_Tgorjachego_vozduha_ED_kanal_1_command : UINT;
    AI_Tgorjachego_vozduha_ED_kanal_1_newHL : LREAL;
    AI_Tgorjachego_vozduha_ED_kanal_1_newLL : LREAL;
    AI_Tgorjachego_vozduha_ED_kanal_1_status : UDINT;
    AI_Tgorjachego_vozduha_ED_kanal_1_value : LREAL;
    AI_Tgorjachego_vozduha_ED_kanal_1_HW : LREAL;
    AI_Tgorjachego_vozduha_ED_kanal_1_newHW : LREAL;
    AI_Tgorjachego_vozduha_ED_kanal_2_HL : LREAL;
    AI_Tgorjachego_vozduha_ED_kanal_2_LL : LREAL;
    AI_Tgorjachego_vozduha_ED_kanal_2_command : UINT;
    AI_Tgorjachego_vozduha_ED_kanal_2_newHL : LREAL;
    AI_Tgorjachego_vozduha_ED_kanal_2_newLL : LREAL;
    AI_Tgorjachego_vozduha_ED_kanal_2_status : UDINT;
    AI_Tgorjachego_vozduha_ED_kanal_2_value : LREAL;
    AI_Tgorjachego_vozduha_ED_kanal_2_HW : LREAL;
    AI_Tgorjachego_vozduha_ED_kanal_2_newHW : LREAL;
    AI_Tnarujnogo_vozduha_HL : LREAL;
    AI_Tnarujnogo_vozduha_LL : LREAL;
    AI_Tnarujnogo_vozduha_command : UINT;
    AI_Tnarujnogo_vozduha_newHL : LREAL;
    AI_Tnarujnogo_vozduha_newLL : LREAL;
    AI_Tnarujnogo_vozduha_status : UDINT;
    AI_Tnarujnogo_vozduha_value : LREAL;
    AI_Tnarujnogo_vozduha_HW : LREAL;
    AI_Tnarujnogo_vozduha_newHW : LREAL;
    AI_Tgaza_na_vhode_H_HL : LREAL;
    AI_Tgaza_na_vhode_H_LL : LREAL;
    AI_Tgaza_na_vhode_H_command : UINT;
    AI_Tgaza_na_vhode_H_newHL : LREAL;
    AI_Tgaza_na_vhode_H_newLL : LREAL;
    AI_Tgaza_na_vhode_H_status : UDINT;
    AI_Tgaza_na_vhode_H_value : LREAL;
    AI_Tgaza_na_vhode_H_HW : LREAL;
    AI_Tgaza_na_vhode_H_newHW : LREAL;
    AI_Tgaza_na_vyhode_H_HL : LREAL;
    AI_Tgaza_na_vyhode_H_LL : LREAL;
    AI_Tgaza_na_vyhode_H_command : UINT;
    AI_Tgaza_na_vyhode_H_newHL : LREAL;
    AI_Tgaza_na_vyhode_H_newLL : LREAL;
    AI_Tgaza_na_vyhode_H_status : UDINT;
    AI_Tgaza_na_vyhode_H_value : LREAL;
    AI_Tgaza_na_vyhode_H_HW : LREAL;
    AI_Tgaza_na_vyhode_H_newHW : LREAL;
    AI_Tgaza_na_vyhode_H_HA : LREAL;
    AI_Tgaza_na_vyhode_H_newHA : LREAL;
    AI_Tmasla_do_AVOM_HL : LREAL;
    AI_Tmasla_do_AVOM_LL : LREAL;
    AI_Tmasla_do_AVOM_command : UINT;
    AI_Tmasla_do_AVOM_newHL : LREAL;
    AI_Tmasla_do_AVOM_newLL : LREAL;
    AI_Tmasla_do_AVOM_status : UDINT;
    AI_Tmasla_do_AVOM_value : LREAL;
    AI_Tmasla_do_AVOM_HW : LREAL;
    AI_Tmasla_do_AVOM_newHW : LREAL;
    AI_Tmasla_posle_AVOM_HL : LREAL;
    AI_Tmasla_posle_AVOM_LL : LREAL;
    AI_Tmasla_posle_AVOM_command : UINT;
    AI_Tmasla_posle_AVOM_newHL : LREAL;
    AI_Tmasla_posle_AVOM_newLL : LREAL;
    AI_Tmasla_posle_AVOM_status : UDINT;
    AI_Tmasla_posle_AVOM_value : LREAL;
    AI_Tmasla_posle_AVOM_HW : LREAL;
    AI_Tmasla_posle_AVOM_newHW : LREAL;
    AI_Tmasla_MB_HL : LREAL;
    AI_Tmasla_MB_LL : LREAL;
    AI_Tmasla_MB_command : UINT;
    AI_Tmasla_MB_newHL : LREAL;
    AI_Tmasla_MB_newLL : LREAL;
    AI_Tmasla_MB_status : UDINT;
    AI_Tmasla_MB_value : LREAL;
    AI_Tmasla_MB_HW : LREAL;
    AI_Tmasla_MB_newHW : LREAL;
    AI_Tmasla_MB_TEN_HL : LREAL;
    AI_Tmasla_MB_TEN_LL : LREAL;
    AI_Tmasla_MB_TEN_command : UINT;
    AI_Tmasla_MB_TEN_newHL : LREAL;
    AI_Tmasla_MB_TEN_newLL : LREAL;
    AI_Tmasla_MB_TEN_status : UDINT;
    AI_Tmasla_MB_TEN_value : LREAL;
    AI_Tmasla_MB_TEN_HW : LREAL;
    AI_Tmasla_MB_TEN_newHW : LREAL;
    AI_Tshu_HL : LREAL;
    AI_Tshu_LL : LREAL;
    AI_Tshu_command : UINT;
    AI_Tshu_newHL : LREAL;
    AI_Tshu_newLL : LREAL;
    AI_Tshu_status : UDINT;
    AI_Tshu_value : LREAL;
    AI_Pmaslo_sm_nizkoe_HL : LREAL;
    AI_Pmaslo_sm_nizkoe_LL : LREAL;
    AI_Pmaslo_sm_nizkoe_command : UINT;
    AI_Pmaslo_sm_nizkoe_newHL : LREAL;
    AI_Pmaslo_sm_nizkoe_newLL : LREAL;
    AI_Pmaslo_sm_nizkoe_status : UDINT;
    AI_Pmaslo_sm_nizkoe_value : LREAL;
    AI_Pmaslo_sm_nizkoe_LW : LREAL;
    AI_Pmaslo_sm_nizkoe_newLW : LREAL;
    AI_Pmaslo_sm_nizkoe_LA : LREAL;
    AI_Pmaslo_sm_nizkoe_newLA : LREAL;
    AI_Pmaslo_sm_vysokoe_HL : LREAL;
    AI_Pmaslo_sm_vysokoe_LL : LREAL;
    AI_Pmaslo_sm_vysokoe_command : UINT;
    AI_Pmaslo_sm_vysokoe_newHL : LREAL;
    AI_Pmaslo_sm_vysokoe_newLL : LREAL;
    AI_Pmaslo_sm_vysokoe_status : UDINT;
    AI_Pmaslo_sm_vysokoe_value : LREAL;
    AI_Pmaslo_sm_vysokoe_LW : LREAL;
    AI_Pmaslo_sm_vysokoe_newLW : LREAL;
    AI_Pmaslo_sm_vysokoe_LA : LREAL;
    AI_Pmaslo_sm_vysokoe_newLA : LREAL;
    AI_Pmasla_posle_GNS_HL : LREAL;
    AI_Pmasla_posle_GNS_LL : LREAL;
    AI_Pmasla_posle_GNS_command : UINT;
    AI_Pmasla_posle_GNS_newHL : LREAL;
    AI_Pmasla_posle_GNS_newLL : LREAL;
    AI_Pmasla_posle_GNS_status : UDINT;
    AI_Pmasla_posle_GNS_value : LREAL;
    AI_Pmasla_posle_GNS_HW : LREAL;
    AI_Pmasla_posle_GNS_newHW : LREAL;
    AI_Pmasla_posle_GNS_LW : LREAL;
    AI_Pmasla_posle_GNS_newLW : LREAL;
    AI_Pmasla_posle_NU_HL : LREAL;
    AI_Pmasla_posle_NU_LL : LREAL;
    AI_Pmasla_posle_NU_command : UINT;
    AI_Pmasla_posle_NU_newHL : LREAL;
    AI_Pmasla_posle_NU_newLL : LREAL;
    AI_Pmasla_posle_NU_status : UDINT;
    AI_Pmasla_posle_NU_value : LREAL;
    AI_Pmasla_posle_NU_LW : LREAL;
    AI_Pmasla_posle_NU_newLW : LREAL;
    AI_Pgaza_na_vhode_nagnetatelia_HL : LREAL;
    AI_Pgaza_na_vhode_nagnetatelia_LL : LREAL;
    AI_Pgaza_na_vhode_nagnetatelia_command : UINT;
    AI_Pgaza_na_vhode_nagnetatelia_newHL : LREAL;
    AI_Pgaza_na_vhode_nagnetatelia_newLL : LREAL;
    AI_Pgaza_na_vhode_nagnetatelia_status : UDINT;
    AI_Pgaza_na_vhode_nagnetatelia_value : LREAL;
    AI_Pgaza_na_vhode_nagnetatelia_LW : LREAL;
    AI_Pgaza_na_vhode_nagnetatelia_newLW : LREAL;
    AI_Pgaza_na_vyhode_nagnetatelia_HL : LREAL;
    AI_Pgaza_na_vyhode_nagnetatelia_LL : LREAL;
    AI_Pgaza_na_vyhode_nagnetatelia_command : UINT;
    AI_Pgaza_na_vyhode_nagnetatelia_newHL : LREAL;
    AI_Pgaza_na_vyhode_nagnetatelia_newLL : LREAL;
    AI_Pgaza_na_vyhode_nagnetatelia_status : UDINT;
    AI_Pgaza_na_vyhode_nagnetatelia_value : LREAL;
    AI_Pgaza_na_vyhode_nagnetatelia_LW : LREAL;
    AI_Pgaza_na_vyhode_nagnetatelia_newLW : LREAL;
    AI_Pgaza_na_vyhode_nagnetatelia_HA : LREAL;
    AI_Pgaza_na_vyhode_nagnetatelia_newHA : LREAL;
    AI_Pimpuls_gaz_HL : LREAL;
    AI_Pimpuls_gaz_LL : LREAL;
    AI_Pimpuls_gaz_command : UINT;
    AI_Pimpuls_gaz_newHL : LREAL;
    AI_Pimpuls_gaz_newLL : LREAL;
    AI_Pimpuls_gaz_status : UDINT;
    AI_Pimpuls_gaz_value : LREAL;
    AI_Pimpuls_gaz_LW : LREAL;
    AI_Pimpuls_gaz_newLW : LREAL;
    AI_dPgaza_na_maslo_filtre_HL : LREAL;
    AI_dPgaza_na_maslo_filtre_LL : LREAL;
    AI_dPgaza_na_maslo_filtre_command : UINT;
    AI_dPgaza_na_maslo_filtre_newHL : LREAL;
    AI_dPgaza_na_maslo_filtre_newLL : LREAL;
    AI_dPgaza_na_maslo_filtre_status : UDINT;
    AI_dPgaza_na_maslo_filtre_value : LREAL;
    AI_dPgaza_na_maslo_filtre_HW : LREAL;
    AI_dPgaza_na_maslo_filtre_newHW : LREAL;
    AI_dPgaza_na_konfuzore_HL : LREAL;
    AI_dPgaza_na_konfuzore_LL : LREAL;
    AI_dPgaza_na_konfuzore_command : UINT;
    AI_dPgaza_na_konfuzore_newHL : LREAL;
    AI_dPgaza_na_konfuzore_newLL : LREAL;
    AI_dPgaza_na_konfuzore_status : UDINT;
    AI_dPgaza_na_konfuzore_value : LREAL;
    AI_dPgaza_na_konfuzore_LW : LREAL;
    AI_dPgaza_na_konfuzore_newLW : LREAL;
    AI_dPmaslo_gaz_HL : LREAL;
    AI_dPmaslo_gaz_LL : LREAL;
    AI_dPmaslo_gaz_command : UINT;
    AI_dPmaslo_gaz_newHL : LREAL;
    AI_dPmaslo_gaz_newLL : LREAL;
    AI_dPmaslo_gaz_status : UDINT;
    AI_dPmaslo_gaz_value : LREAL;
    AI_dPmaslo_gaz_LW : LREAL;
    AI_dPmaslo_gaz_newLW : LREAL;
    AI_dPmaslo_gaz_LA : LREAL;
    AI_dPmaslo_gaz_newLA : LREAL;
    AI_Os_sdvig_nagnetatelja_plus_HL : LREAL;
    AI_Os_sdvig_nagnetatelja_plus_LL : LREAL;
    AI_Os_sdvig_nagnetatelja_plus_command : UINT;
    AI_Os_sdvig_nagnetatelja_plus_newHL : LREAL;
    AI_Os_sdvig_nagnetatelja_plus_newLL : LREAL;
    AI_Os_sdvig_nagnetatelja_plus_status : UDINT;
    AI_Os_sdvig_nagnetatelja_plus_value : LREAL;
    AI_Os_sdvig_nagnetatelja_plus_HW : LREAL;
    AI_Os_sdvig_nagnetatelja_plus_newHW : LREAL;
    AI_Os_sdvig_nagnetatelja_plus_HA : LREAL;
    AI_Os_sdvig_nagnetatelja_plus_newHA : LREAL;
    AI_Os_sdvig_nagnetatelja_minus_HL : LREAL;
    AI_Os_sdvig_nagnetatelja_minus_LL : LREAL;
    AI_Os_sdvig_nagnetatelja_minus_command : UINT;
    AI_Os_sdvig_nagnetatelja_minus_newHL : LREAL;
    AI_Os_sdvig_nagnetatelja_minus_newLL : LREAL;
    AI_Os_sdvig_nagnetatelja_minus_status : UDINT;
    AI_Os_sdvig_nagnetatelja_minus_value : LREAL;
    AI_Os_sdvig_nagnetatelja_minus_LW : LREAL;
    AI_Os_sdvig_nagnetatelja_minus_newLW : LREAL;
    AI_Os_sdvig_nagnetatelja_minus_LA : LREAL;
    AI_Os_sdvig_nagnetatelja_minus_newLA : LREAL;
    AI_Yroven_masla_MB_HL : LREAL;
    AI_Yroven_masla_MB_LL : LREAL;
    AI_Yroven_masla_MB_command : UINT;
    AI_Yroven_masla_MB_newHL : LREAL;
    AI_Yroven_masla_MB_newLL : LREAL;
    AI_Yroven_masla_MB_status : UDINT;
    AI_Yroven_masla_MB_value : LREAL;
    AI_Yroven_masla_MB_LW : LREAL;
    AI_Yroven_masla_MB_newLW : LREAL;
    AI_Kontrol_per_220V_HL : LREAL;
    AI_Kontrol_per_220V_LL : LREAL;
    AI_Kontrol_per_220V_command : UINT;
    AI_Kontrol_per_220V_newHL : LREAL;
    AI_Kontrol_per_220V_newLL : LREAL;
    AI_Kontrol_per_220V_status : UDINT;
    AI_Kontrol_per_220V_value : LREAL;
    AI_Kontrol_per_220V_HW : LREAL;
    AI_Kontrol_per_220V_newHW : LREAL;
    AI_Kontrol_per_220V_LW : LREAL;
    AI_Kontrol_per_220V_newLW : LREAL;
    AI_Kontrol_post_220V_HL : LREAL;
    AI_Kontrol_post_220V_LL : LREAL;
    AI_Kontrol_post_220V_command : UINT;
    AI_Kontrol_post_220V_newHL : LREAL;
    AI_Kontrol_post_220V_newLL : LREAL;
    AI_Kontrol_post_220V_status : UDINT;
    AI_Kontrol_post_220V_value : LREAL;
    AI_Kontrol_post_220V_HW : LREAL;
    AI_Kontrol_post_220V_newHW : LREAL;
    AI_Kontrol_post_220V_LW : LREAL;
    AI_Kontrol_post_220V_newLW : LREAL;
    AI_Tok_statora_HL : LREAL;
    AI_Tok_statora_LL : LREAL;
    AI_Tok_statora_command : UINT;
    AI_Tok_statora_newHL : LREAL;
    AI_Tok_statora_newLL : LREAL;
    AI_Tok_statora_status : UDINT;
    AI_Tok_statora_value : LREAL;
    AI_Tok_statora_LW : LREAL;
    AI_Tok_statora_newLW : LREAL;
    AI_Vibro_skorost_OPED_T1_HL : LREAL;
    AI_Vibro_skorost_OPED_T1_LL : LREAL;
    AI_Vibro_skorost_OPED_T1_command : UINT;
    AI_Vibro_skorost_OPED_T1_newHL : LREAL;
    AI_Vibro_skorost_OPED_T1_newLL : LREAL;
    AI_Vibro_skorost_OPED_T1_status : UDINT;
    AI_Vibro_skorost_OPED_T1_value : LREAL;
    AI_Vibro_skorost_OPED_T1_HW : LREAL;
    AI_Vibro_skorost_OPED_T1_newHW : LREAL;
    AI_Vibro_skorost_OPED_T1_HA : LREAL;
    AI_Vibro_skorost_OPED_T1_newHA : LREAL;
    AI_Vibro_skorost_OYPED_T2_HL : LREAL;
    AI_Vibro_skorost_OYPED_T2_LL : LREAL;
    AI_Vibro_skorost_OYPED_T2_command : UINT;
    AI_Vibro_skorost_OYPED_T2_newHL : LREAL;
    AI_Vibro_skorost_OYPED_T2_newLL : LREAL;
    AI_Vibro_skorost_OYPED_T2_status : UDINT;
    AI_Vibro_skorost_OYPED_T2_value : LREAL;
    AI_Vibro_skorost_OYPED_T2_HW : LREAL;
    AI_Vibro_skorost_OYPED_T2_newHW : LREAL;
    AI_Vibro_skorost_OYPED_T2_HA : LREAL;
    AI_Vibro_skorost_OYPED_T2_newHA : LREAL;
    AI_Vibro_skorost_OYP_kolesa_ED_T3_HL : LREAL;
    AI_Vibro_skorost_OYP_kolesa_ED_T3_LL : LREAL;
    AI_Vibro_skorost_OYP_kolesa_ED_T3_command : UINT;
    AI_Vibro_skorost_OYP_kolesa_ED_T3_newHL : LREAL;
    AI_Vibro_skorost_OYP_kolesa_ED_T3_newLL : LREAL;
    AI_Vibro_skorost_OYP_kolesa_ED_T3_status : UDINT;
    AI_Vibro_skorost_OYP_kolesa_ED_T3_value : LREAL;
    AI_Vibro_skorost_OYP_kolesa_ED_T3_HW : LREAL;
    AI_Vibro_skorost_OYP_kolesa_ED_T3_newHW : LREAL;
    AI_Vibro_skorost_OYP_kolesa_ED_T3_HA : LREAL;
    AI_Vibro_skorost_OYP_kolesa_ED_T3_newHA : LREAL;
    AI_Vibro_skorost_OP_kolesa_RH_T4_HL : LREAL;
    AI_Vibro_skorost_OP_kolesa_RH_T4_LL : LREAL;
    AI_Vibro_skorost_OP_kolesa_RH_T4_command : UINT;
    AI_Vibro_skorost_OP_kolesa_RH_T4_newHL : LREAL;
    AI_Vibro_skorost_OP_kolesa_RH_T4_newLL : LREAL;
    AI_Vibro_skorost_OP_kolesa_RH_T4_status : UDINT;
    AI_Vibro_skorost_OP_kolesa_RH_T4_value : LREAL;
    AI_Vibro_skorost_OP_kolesa_RH_T4_HW : LREAL;
    AI_Vibro_skorost_OP_kolesa_RH_T4_newHW : LREAL;
    AI_Vibro_skorost_OP_kolesa_RH_T4_HA : LREAL;
    AI_Vibro_skorost_OP_kolesa_RH_T4_newHA : LREAL;
    AI_Vibro_skorost_OP_shesterni_RED_T5_HL : LREAL;
    AI_Vibro_skorost_OP_shesterni_RED_T5_LL : LREAL;
    AI_Vibro_skorost_OP_shesterni_RED_T5_command : UINT;
    AI_Vibro_skorost_OP_shesterni_RED_T5_newHL : LREAL;
    AI_Vibro_skorost_OP_shesterni_RED_T5_newLL : LREAL;
    AI_Vibro_skorost_OP_shesterni_RED_T5_status : UDINT;
    AI_Vibro_skorost_OP_shesterni_RED_T5_value : LREAL;
    AI_Vibro_skorost_OP_shesterni_RED_T5_HW : LREAL;
    AI_Vibro_skorost_OP_shesterni_RED_T5_newHW : LREAL;
    AI_Vibro_skorost_OP_shesterni_RED_T5_HA : LREAL;
    AI_Vibro_skorost_OP_shesterni_RED_T5_newHA : LREAL;
    AI_Vibro_skorost_OP_shesterni_RED_T6_HL : LREAL;
    AI_Vibro_skorost_OP_shesterni_RED_T6_LL : LREAL;
    AI_Vibro_skorost_OP_shesterni_RED_T6_command : UINT;
    AI_Vibro_skorost_OP_shesterni_RED_T6_newHL : LREAL;
    AI_Vibro_skorost_OP_shesterni_RED_T6_newLL : LREAL;
    AI_Vibro_skorost_OP_shesterni_RED_T6_status : UDINT;
    AI_Vibro_skorost_OP_shesterni_RED_T6_value : LREAL;
    AI_Vibro_skorost_OP_shesterni_RED_T6_HW : LREAL;
    AI_Vibro_skorost_OP_shesterni_RED_T6_newHW : LREAL;
    AI_Vibro_skorost_OP_shesterni_RED_T6_HA : LREAL;
    AI_Vibro_skorost_OP_shesterni_RED_T6_newHA : LREAL;
  END_VAR

  AI_Tstali_statora_kanal_1_HL := ai.Tstali_statora_kanal_1.HL;
  AI_Tstali_statora_kanal_1_LL := ai.Tstali_statora_kanal_1.LL;
  AI_Tstali_statora_kanal_1_newHL := ai.Tstali_statora_kanal_1.dHL;
  AI_Tstali_statora_kanal_1_newLL := ai.Tstali_statora_kanal_1.dLL;
  AI_Tstali_statora_kanal_1_HW := ai.Tstali_statora_kanal_1.HW;
  AI_Tstali_statora_kanal_1_newHW := ai.Tstali_statora_kanal_1.dHW;

  AI_Tstali_statora_kanal_2_HL := ai.Tstali_statora_kanal_2.HL;
  AI_Tstali_statora_kanal_2_LL := ai.Tstali_statora_kanal_2.LL;
  AI_Tstali_statora_kanal_2_newHL := ai.Tstali_statora_kanal_2.dHL;
  AI_Tstali_statora_kanal_2_newLL := ai.Tstali_statora_kanal_2.dLL;
  AI_Tstali_statora_kanal_2_HW := ai.Tstali_statora_kanal_2.HW;
  AI_Tstali_statora_kanal_2_newHW := ai.Tstali_statora_kanal_2.dHW;

  AI_Tstali_statora_kanal_3_HL := ai.Tstali_statora_kanal_3.HL;
  AI_Tstali_statora_kanal_3_LL := ai.Tstali_statora_kanal_3.LL;
  AI_Tstali_statora_kanal_3_newHL := ai.Tstali_statora_kanal_3.dHL;
  AI_Tstali_statora_kanal_3_newLL := ai.Tstali_statora_kanal_3.dLL;
  AI_Tstali_statora_kanal_3_HW := ai.Tstali_statora_kanal_3.HW;
  AI_Tstali_statora_kanal_3_newHW := ai.Tstali_statora_kanal_3.dHW;

  AI_Tmedi_statora_kanal_1_HL := ai.Tmedi_statora_kanal_1.HL;
  AI_Tmedi_statora_kanal_1_LL := ai.Tmedi_statora_kanal_1.LL;
  AI_Tmedi_statora_kanal_1_newHL := ai.Tmedi_statora_kanal_1.dHL;
  AI_Tmedi_statora_kanal_1_newLL := ai.Tmedi_statora_kanal_1.dLL;
  AI_Tmedi_statora_kanal_1_HW := ai.Tmedi_statora_kanal_1.HW;
  AI_Tmedi_statora_kanal_1_newHW := ai.Tmedi_statora_kanal_1.dHW;

  AI_Tmedi_statora_kanal_2_HL := ai.Tmedi_statora_kanal_2.HL;
  AI_Tmedi_statora_kanal_2_LL := ai.Tmedi_statora_kanal_2.LL;
  AI_Tmedi_statora_kanal_2_newHL := ai.Tmedi_statora_kanal_2.dHL;
  AI_Tmedi_statora_kanal_2_newLL := ai.Tmedi_statora_kanal_2.dLL;
  AI_Tmedi_statora_kanal_2_HW := ai.Tmedi_statora_kanal_2.HW;
  AI_Tmedi_statora_kanal_2_newHW := ai.Tmedi_statora_kanal_2.dHW;

  AI_Tmedi_statora_kanal_3_HL := ai.Tmedi_statora_kanal_3.HL;
  AI_Tmedi_statora_kanal_3_LL := ai.Tmedi_statora_kanal_3.LL;
  AI_Tmedi_statora_kanal_3_newHL := ai.Tmedi_statora_kanal_3.dHL;
  AI_Tmedi_statora_kanal_3_newLL := ai.Tmedi_statora_kanal_3.dLL;
  AI_Tmedi_statora_kanal_3_HW := ai.Tmedi_statora_kanal_3.HW;
  AI_Tmedi_statora_kanal_3_newHW := ai.Tmedi_statora_kanal_3.dHW;

  AI_Toporno_podshipnika_EDT_1_HL := ai.Toporno_podshipnika_EDT_1.HL;
  AI_Toporno_podshipnika_EDT_1_LL := ai.Toporno_podshipnika_EDT_1.LL;
  AI_Toporno_podshipnika_EDT_1_newHL := ai.Toporno_podshipnika_EDT_1.dHL;
  AI_Toporno_podshipnika_EDT_1_newLL := ai.Toporno_podshipnika_EDT_1.dLL;
  AI_Toporno_podshipnika_EDT_1_HW := ai.Toporno_podshipnika_EDT_1.HW;
  AI_Toporno_podshipnika_EDT_1_newHW := ai.Toporno_podshipnika_EDT_1.dHW;
  AI_Toporno_podshipnika_EDT_1_HA := ai.Toporno_podshipnika_EDT_1.HA;
  AI_Toporno_podshipnika_EDT_1_newHA := ai.Toporno_podshipnika_EDT_1.dHA;

  AI_Toy_podshipnika_EDT_2_HL := ai.Toy_podshipnika_EDT_2.HL;
  AI_Toy_podshipnika_EDT_2_LL := ai.Toy_podshipnika_EDT_2.LL;
  AI_Toy_podshipnika_EDT_2_newHL := ai.Toy_podshipnika_EDT_2.dHL;
  AI_Toy_podshipnika_EDT_2_newLL := ai.Toy_podshipnika_EDT_2.dLL;
  AI_Toy_podshipnika_EDT_2_HW := ai.Toy_podshipnika_EDT_2.HW;
  AI_Toy_podshipnika_EDT_2_newHW := ai.Toy_podshipnika_EDT_2.dHW;
  AI_Toy_podshipnika_EDT_2_HA := ai.Toy_podshipnika_EDT_2.HA;
  AI_Toy_podshipnika_EDT_2_newHA := ai.Toy_podshipnika_EDT_2.dHA;

  AI_Toy_podshipnika_kol_EDT_3_HL := ai.Toy_podshipnika_kol_EDT_3.HL;
  AI_Toy_podshipnika_kol_EDT_3_LL := ai.Toy_podshipnika_kol_EDT_3.LL;
  AI_Toy_podshipnika_kol_EDT_3_newHL := ai.Toy_podshipnika_kol_EDT_3.dHL;
  AI_Toy_podshipnika_kol_EDT_3_newLL := ai.Toy_podshipnika_kol_EDT_3.dLL;
  AI_Toy_podshipnika_kol_EDT_3_HW := ai.Toy_podshipnika_kol_EDT_3.HW;
  AI_Toy_podshipnika_kol_EDT_3_newHW := ai.Toy_podshipnika_kol_EDT_3.dHW;
  AI_Toy_podshipnika_kol_EDT_3_HA := ai.Toy_podshipnika_kol_EDT_3.HA;
  AI_Toy_podshipnika_kol_EDT_3_newHA := ai.Toy_podshipnika_kol_EDT_3.dHA;

  AI_Toy_podshipnika_kol_EDT_4_HL := ai.Toy_podshipnika_kol_EDT_4.HL;
  AI_Toy_podshipnika_kol_EDT_4_LL := ai.Toy_podshipnika_kol_EDT_4.LL;
  AI_Toy_podshipnika_kol_EDT_4_newHL := ai.Toy_podshipnika_kol_EDT_4.dHL;
  AI_Toy_podshipnika_kol_EDT_4_newLL := ai.Toy_podshipnika_kol_EDT_4.dLL;
  AI_Toy_podshipnika_kol_EDT_4_HW := ai.Toy_podshipnika_kol_EDT_4.HW;
  AI_Toy_podshipnika_kol_EDT_4_newHW := ai.Toy_podshipnika_kol_EDT_4.dHW;
  AI_Toy_podshipnika_kol_EDT_4_HA := ai.Toy_podshipnika_kol_EDT_4.HA;
  AI_Toy_podshipnika_kol_EDT_4_newHA := ai.Toy_podshipnika_kol_EDT_4.dHA;

  AI_Toy_podshipnika_shest_red_EDT_5_HL := ai.Toy_podshipnika_shest_red_EDT_5.HL;
  AI_Toy_podshipnika_shest_red_EDT_5_LL := ai.Toy_podshipnika_shest_red_EDT_5.LL;
  AI_Toy_podshipnika_shest_red_EDT_5_newHL := ai.Toy_podshipnika_shest_red_EDT_5.dHL;
  AI_Toy_podshipnika_shest_red_EDT_5_newLL := ai.Toy_podshipnika_shest_red_EDT_5.dLL;
  AI_Toy_podshipnika_shest_red_EDT_5_HW := ai.Toy_podshipnika_shest_red_EDT_5.HW;
  AI_Toy_podshipnika_shest_red_EDT_5_newHW := ai.Toy_podshipnika_shest_red_EDT_5.dHW;
  AI_Toy_podshipnika_shest_red_EDT_5_HA := ai.Toy_podshipnika_shest_red_EDT_5.HA;
  AI_Toy_podshipnika_shest_red_EDT_5_newHA := ai.Toy_podshipnika_shest_red_EDT_5.dHA;

  AI_Ty_podshipnika_red_EDT_6_HL := ai.Ty_podshipnika_red_EDT_6.HL;
  AI_Ty_podshipnika_red_EDT_6_LL := ai.Ty_podshipnika_red_EDT_6.LL;
  AI_Ty_podshipnika_red_EDT_6_newHL := ai.Ty_podshipnika_red_EDT_6.dHL;
  AI_Ty_podshipnika_red_EDT_6_newLL := ai.Ty_podshipnika_red_EDT_6.dLL;
  AI_Ty_podshipnika_red_EDT_6_HW := ai.Ty_podshipnika_red_EDT_6.HW;
  AI_Ty_podshipnika_red_EDT_6_newHW := ai.Ty_podshipnika_red_EDT_6.dHW;
  AI_Ty_podshipnika_red_EDT_6_HA := ai.Ty_podshipnika_red_EDT_6.HA;
  AI_Ty_podshipnika_red_EDT_6_newHA := ai.Ty_podshipnika_red_EDT_6.dHA;

  AI_Ty_podshipnika_nagnet_EDT_7_1_HL := ai.Ty_podshipnika_nagnet_EDT_7_1.HL;
  AI_Ty_podshipnika_nagnet_EDT_7_1_LL := ai.Ty_podshipnika_nagnet_EDT_7_1.LL;
  AI_Ty_podshipnika_nagnet_EDT_7_1_newHL := ai.Ty_podshipnika_nagnet_EDT_7_1.dHL;
  AI_Ty_podshipnika_nagnet_EDT_7_1_newLL := ai.Ty_podshipnika_nagnet_EDT_7_1.dLL;
  AI_Ty_podshipnika_nagnet_EDT_7_1_HW := ai.Ty_podshipnika_nagnet_EDT_7_1.HW;
  AI_Ty_podshipnika_nagnet_EDT_7_1_newHW := ai.Ty_podshipnika_nagnet_EDT_7_1.dHW;
  AI_Ty_podshipnika_nagnet_EDT_7_1_HA := ai.Ty_podshipnika_nagnet_EDT_7_1.HA;
  AI_Ty_podshipnika_nagnet_EDT_7_1_newHA := ai.Ty_podshipnika_nagnet_EDT_7_1.dHA;

  AI_Ty_podshipnika_nagnet_EDT_7_2_HL := ai.Ty_podshipnika_nagnet_EDT_7_2.HL;
  AI_Ty_podshipnika_nagnet_EDT_7_2_LL := ai.Ty_podshipnika_nagnet_EDT_7_2.LL;
  AI_Ty_podshipnika_nagnet_EDT_7_2_newHL := ai.Ty_podshipnika_nagnet_EDT_7_2.dHL;
  AI_Ty_podshipnika_nagnet_EDT_7_2_newLL := ai.Ty_podshipnika_nagnet_EDT_7_2.dLL;
  AI_Ty_podshipnika_nagnet_EDT_7_2_HW := ai.Ty_podshipnika_nagnet_EDT_7_2.HW;
  AI_Ty_podshipnika_nagnet_EDT_7_2_newHW := ai.Ty_podshipnika_nagnet_EDT_7_2.dHW;
  AI_Ty_podshipnika_nagnet_EDT_7_2_HA := ai.Ty_podshipnika_nagnet_EDT_7_2.HA;
  AI_Ty_podshipnika_nagnet_EDT_7_2_newHA := ai.Ty_podshipnika_nagnet_EDT_7_2.dHA;

  AI_Toy_podshipnika_svobod_konca_EDT_8_1_HL := ai.Toy_podshipnika_svobod_konca_EDT_8_1.HL;
  AI_Toy_podshipnika_svobod_konca_EDT_8_1_LL := ai.Toy_podshipnika_svobod_konca_EDT_8_1.LL;
  AI_Toy_podshipnika_svobod_konca_EDT_8_1_newHL := ai.Toy_podshipnika_svobod_konca_EDT_8_1.dHL;
  AI_Toy_podshipnika_svobod_konca_EDT_8_1_newLL := ai.Toy_podshipnika_svobod_konca_EDT_8_1.dLL;
  AI_Toy_podshipnika_svobod_konca_EDT_8_1_HW := ai.Toy_podshipnika_svobod_konca_EDT_8_1.HW;
  AI_Toy_podshipnika_svobod_konca_EDT_8_1_newHW := ai.Toy_podshipnika_svobod_konca_EDT_8_1.dHW;
  AI_Toy_podshipnika_svobod_konca_EDT_8_1_HA := ai.Toy_podshipnika_svobod_konca_EDT_8_1.HA;
  AI_Toy_podshipnika_svobod_konca_EDT_8_1_newHA := ai.Toy_podshipnika_svobod_konca_EDT_8_1.dHA;

  AI_Toy_podshipnika_svobod_konca_EDT_8_2_HL := ai.Toy_podshipnika_svobod_konca_EDT_8_2.HL;
  AI_Toy_podshipnika_svobod_konca_EDT_8_2_LL := ai.Toy_podshipnika_svobod_konca_EDT_8_2.LL;
  AI_Toy_podshipnika_svobod_konca_EDT_8_2_newHL := ai.Toy_podshipnika_svobod_konca_EDT_8_2.dHL;
  AI_Toy_podshipnika_svobod_konca_EDT_8_2_newLL := ai.Toy_podshipnika_svobod_konca_EDT_8_2.dLL;
  AI_Toy_podshipnika_svobod_konca_EDT_8_2_HW := ai.Toy_podshipnika_svobod_konca_EDT_8_2.HW;
  AI_Toy_podshipnika_svobod_konca_EDT_8_2_newHW := ai.Toy_podshipnika_svobod_konca_EDT_8_2.dHW;
  AI_Toy_podshipnika_svobod_konca_EDT_8_2_HA := ai.Toy_podshipnika_svobod_konca_EDT_8_2.HA;
  AI_Toy_podshipnika_svobod_konca_EDT_8_2_newHA := ai.Toy_podshipnika_svobod_konca_EDT_8_2.dHA;

  AI_Toy_podshipnika_rab_kol_EDT_9_1_HL := ai.Toy_podshipnika_rab_kol_EDT_9_1.HL;
  AI_Toy_podshipnika_rab_kol_EDT_9_1_LL := ai.Toy_podshipnika_rab_kol_EDT_9_1.LL;
  AI_Toy_podshipnika_rab_kol_EDT_9_1_newHL := ai.Toy_podshipnika_rab_kol_EDT_9_1.dHL;
  AI_Toy_podshipnika_rab_kol_EDT_9_1_newLL := ai.Toy_podshipnika_rab_kol_EDT_9_1.dLL;
  AI_Toy_podshipnika_rab_kol_EDT_9_1_HW := ai.Toy_podshipnika_rab_kol_EDT_9_1.HW;
  AI_Toy_podshipnika_rab_kol_EDT_9_1_newHW := ai.Toy_podshipnika_rab_kol_EDT_9_1.dHW;
  AI_Toy_podshipnika_rab_kol_EDT_9_1_HA := ai.Toy_podshipnika_rab_kol_EDT_9_1.HA;
  AI_Toy_podshipnika_rab_kol_EDT_9_1_newHA := ai.Toy_podshipnika_rab_kol_EDT_9_1.dHA;

  AI_Toy_podshipnika_rab_kol_EDT_9_2_HL := ai.Toy_podshipnika_rab_kol_EDT_9_2.HL;
  AI_Toy_podshipnika_rab_kol_EDT_9_2_LL := ai.Toy_podshipnika_rab_kol_EDT_9_2.LL;
  AI_Toy_podshipnika_rab_kol_EDT_9_2_newHL := ai.Toy_podshipnika_rab_kol_EDT_9_2.dHL;
  AI_Toy_podshipnika_rab_kol_EDT_9_2_newLL := ai.Toy_podshipnika_rab_kol_EDT_9_2.dLL;
  AI_Toy_podshipnika_rab_kol_EDT_9_2_HW := ai.Toy_podshipnika_rab_kol_EDT_9_2.HW;
  AI_Toy_podshipnika_rab_kol_EDT_9_2_newHW := ai.Toy_podshipnika_rab_kol_EDT_9_2.dHW;
  AI_Toy_podshipnika_rab_kol_EDT_9_2_HA := ai.Toy_podshipnika_rab_kol_EDT_9_2.HA;
  AI_Toy_podshipnika_rab_kol_EDT_9_2_newHA := ai.Toy_podshipnika_rab_kol_EDT_9_2.dHA;

  AI_Toy_podshipnika_nerab_kol_EDT_10_1_HL := ai.Toy_podshipnika_nerab_kol_EDT_10_1.HL;
  AI_Toy_podshipnika_nerab_kol_EDT_10_1_LL := ai.Toy_podshipnika_nerab_kol_EDT_10_1.LL;
  AI_Toy_podshipnika_nerab_kol_EDT_10_1_newHL := ai.Toy_podshipnika_nerab_kol_EDT_10_1.dHL;
  AI_Toy_podshipnika_nerab_kol_EDT_10_1_newLL := ai.Toy_podshipnika_nerab_kol_EDT_10_1.dLL;
  AI_Toy_podshipnika_nerab_kol_EDT_10_1_HW := ai.Toy_podshipnika_nerab_kol_EDT_10_1.HW;
  AI_Toy_podshipnika_nerab_kol_EDT_10_1_newHW := ai.Toy_podshipnika_nerab_kol_EDT_10_1.dHW;
  AI_Toy_podshipnika_nerab_kol_EDT_10_1_HA := ai.Toy_podshipnika_nerab_kol_EDT_10_1.HA;
  AI_Toy_podshipnika_nerab_kol_EDT_10_1_newHA := ai.Toy_podshipnika_nerab_kol_EDT_10_1.dHA;

  AI_Toy_podshipnika_nerab_kol_EDT_10_2_HL := ai.Toy_podshipnika_nerab_kol_EDT_10_2.HL;
  AI_Toy_podshipnika_nerab_kol_EDT_10_2_LL := ai.Toy_podshipnika_nerab_kol_EDT_10_2.LL;
  AI_Toy_podshipnika_nerab_kol_EDT_10_2_newHL := ai.Toy_podshipnika_nerab_kol_EDT_10_2.dHL;
  AI_Toy_podshipnika_nerab_kol_EDT_10_2_newLL := ai.Toy_podshipnika_nerab_kol_EDT_10_2.dLL;
  AI_Toy_podshipnika_nerab_kol_EDT_10_2_HW := ai.Toy_podshipnika_nerab_kol_EDT_10_2.HW;
  AI_Toy_podshipnika_nerab_kol_EDT_10_2_newHW := ai.Toy_podshipnika_nerab_kol_EDT_10_2.dHW;
  AI_Toy_podshipnika_nerab_kol_EDT_10_2_HA := ai.Toy_podshipnika_nerab_kol_EDT_10_2.HA;
  AI_Toy_podshipnika_nerab_kol_EDT_10_2_newHA := ai.Toy_podshipnika_nerab_kol_EDT_10_2.dHA;

  AI_Tholodnogo_vozduha_ED_kanal_1_HL := ai.Tholodnogo_vozduha_ED_kanal_1.HL;
  AI_Tholodnogo_vozduha_ED_kanal_1_LL := ai.Tholodnogo_vozduha_ED_kanal_1.LL;
  AI_Tholodnogo_vozduha_ED_kanal_1_newHL := ai.Tholodnogo_vozduha_ED_kanal_1.dHL;
  AI_Tholodnogo_vozduha_ED_kanal_1_newLL := ai.Tholodnogo_vozduha_ED_kanal_1.dLL;
  AI_Tholodnogo_vozduha_ED_kanal_1_HW := ai.Tholodnogo_vozduha_ED_kanal_1.HW;
  AI_Tholodnogo_vozduha_ED_kanal_1_newHW := ai.Tholodnogo_vozduha_ED_kanal_1.dHW;

  AI_Tholodnogo_vozduha_ED_kanal_2_HL := ai.Tholodnogo_vozduha_ED_kanal_2.HL;
  AI_Tholodnogo_vozduha_ED_kanal_2_LL := ai.Tholodnogo_vozduha_ED_kanal_2.LL;
  AI_Tholodnogo_vozduha_ED_kanal_2_newHL := ai.Tholodnogo_vozduha_ED_kanal_2.dHL;
  AI_Tholodnogo_vozduha_ED_kanal_2_newLL := ai.Tholodnogo_vozduha_ED_kanal_2.dLL;
  AI_Tholodnogo_vozduha_ED_kanal_2_HW := ai.Tholodnogo_vozduha_ED_kanal_2.HW;
  AI_Tholodnogo_vozduha_ED_kanal_2_newHW := ai.Tholodnogo_vozduha_ED_kanal_2.dHW;

  AI_Tgorjachego_vozduha_ED_kanal_1_HL := ai.Tgorjachego_vozduha_ED_kanal_1.HL;
  AI_Tgorjachego_vozduha_ED_kanal_1_LL := ai.Tgorjachego_vozduha_ED_kanal_1.LL;
  AI_Tgorjachego_vozduha_ED_kanal_1_newHL := ai.Tgorjachego_vozduha_ED_kanal_1.dHL;
  AI_Tgorjachego_vozduha_ED_kanal_1_newLL := ai.Tgorjachego_vozduha_ED_kanal_1.dLL;
  AI_Tgorjachego_vozduha_ED_kanal_1_HW := ai.Tgorjachego_vozduha_ED_kanal_1.HW;
  AI_Tgorjachego_vozduha_ED_kanal_1_newHW := ai.Tgorjachego_vozduha_ED_kanal_1.dHW;

  AI_Tgorjachego_vozduha_ED_kanal_2_HL := ai.Tgorjachego_vozduha_ED_kanal_2.HL;
  AI_Tgorjachego_vozduha_ED_kanal_2_LL := ai.Tgorjachego_vozduha_ED_kanal_2.LL;
  AI_Tgorjachego_vozduha_ED_kanal_2_newHL := ai.Tgorjachego_vozduha_ED_kanal_2.dHL;
  AI_Tgorjachego_vozduha_ED_kanal_2_newLL := ai.Tgorjachego_vozduha_ED_kanal_2.dLL;
  AI_Tgorjachego_vozduha_ED_kanal_2_HW := ai.Tgorjachego_vozduha_ED_kanal_2.HW;
  AI_Tgorjachego_vozduha_ED_kanal_2_newHW := ai.Tgorjachego_vozduha_ED_kanal_2.dHW;

  AI_Tnarujnogo_vozduha_HL := ai.Tnarujnogo_vozduha.HL;
  AI_Tnarujnogo_vozduha_LL := ai.Tnarujnogo_vozduha.LL;
  AI_Tnarujnogo_vozduha_newHL := ai.Tnarujnogo_vozduha.dHL;
  AI_Tnarujnogo_vozduha_newLL := ai.Tnarujnogo_vozduha.dLL;
  AI_Tnarujnogo_vozduha_HW := ai.Tnarujnogo_vozduha.HW;
  AI_Tnarujnogo_vozduha_newHW := ai.Tnarujnogo_vozduha.dHW;

  AI_Tgaza_na_vhode_H_HL := ai.Tgaza_na_vhode_H.HL;
  AI_Tgaza_na_vhode_H_LL := ai.Tgaza_na_vhode_H.LL;
  AI_Tgaza_na_vhode_H_newHL := ai.Tgaza_na_vhode_H.dHL;
  AI_Tgaza_na_vhode_H_newLL := ai.Tgaza_na_vhode_H.dLL;
  AI_Tgaza_na_vhode_H_HW := ai.Tgaza_na_vhode_H.HW;
  AI_Tgaza_na_vhode_H_newHW := ai.Tgaza_na_vhode_H.dHW;

  AI_Tgaza_na_vyhode_H_HL := ai.Tgaza_na_vyhode_H.HL;
  AI_Tgaza_na_vyhode_H_LL := ai.Tgaza_na_vyhode_H.LL;
  AI_Tgaza_na_vyhode_H_newHL := ai.Tgaza_na_vyhode_H.dHL;
  AI_Tgaza_na_vyhode_H_newLL := ai.Tgaza_na_vyhode_H.dLL;
  AI_Tgaza_na_vyhode_H_HW := ai.Tgaza_na_vyhode_H.HW;
  AI_Tgaza_na_vyhode_H_newHW := ai.Tgaza_na_vyhode_H.dHW;
  AI_Tgaza_na_vyhode_H_HA := ai.Tgaza_na_vyhode_H.HA;
  AI_Tgaza_na_vyhode_H_newHA := ai.Tgaza_na_vyhode_H.dHA;

  AI_Tmasla_do_AVOM_HL := ai.Tmasla_do_AVOM.HL;
  AI_Tmasla_do_AVOM_LL := ai.Tmasla_do_AVOM.LL;
  AI_Tmasla_do_AVOM_newHL := ai.Tmasla_do_AVOM.dHL;
  AI_Tmasla_do_AVOM_newLL := ai.Tmasla_do_AVOM.dLL;
  AI_Tmasla_do_AVOM_HW := ai.Tmasla_do_AVOM.HW;
  AI_Tmasla_do_AVOM_newHW := ai.Tmasla_do_AVOM.dHW;

  AI_Tmasla_posle_AVOM_HL := ai.Tmasla_posle_AVOM.HL;
  AI_Tmasla_posle_AVOM_LL := ai.Tmasla_posle_AVOM.LL;
  AI_Tmasla_posle_AVOM_newHL := ai.Tmasla_posle_AVOM.dHL;
  AI_Tmasla_posle_AVOM_newLL := ai.Tmasla_posle_AVOM.dLL;
  AI_Tmasla_posle_AVOM_HW := ai.Tmasla_posle_AVOM.HW;
  AI_Tmasla_posle_AVOM_newHW := ai.Tmasla_posle_AVOM.dHW;

  AI_Tmasla_MB_HL := ai.Tmasla_MB.HL;
  AI_Tmasla_MB_LL := ai.Tmasla_MB.LL;
  AI_Tmasla_MB_newHL := ai.Tmasla_MB.dHL;
  AI_Tmasla_MB_newLL := ai.Tmasla_MB.dLL;
  AI_Tmasla_MB_HW := ai.Tmasla_MB.HW;
  AI_Tmasla_MB_newHW := ai.Tmasla_MB.dHW;

  AI_Tmasla_MB_TEN_HL := ai.Tmasla_MB_TEN.HL;
  AI_Tmasla_MB_TEN_LL := ai.Tmasla_MB_TEN.LL;
  AI_Tmasla_MB_TEN_newHL := ai.Tmasla_MB_TEN.dHL;
  AI_Tmasla_MB_TEN_newLL := ai.Tmasla_MB_TEN.dLL;
  AI_Tmasla_MB_TEN_HW := ai.Tmasla_MB_TEN.HW;
  AI_Tmasla_MB_TEN_newHW := ai.Tmasla_MB_TEN.dHW;

  AI_Tshu_HL := ai.Tshu.HL;
  AI_Tshu_LL := ai.Tshu.LL;
  AI_Tshu_newHL := ai.Tshu.dHL;
  AI_Tshu_newLL := ai.Tshu.dLL;

  AI_Pmaslo_sm_nizkoe_HL := ai.Pmaslo_sm_nizkoe.HL;
  AI_Pmaslo_sm_nizkoe_LL := ai.Pmaslo_sm_nizkoe.LL;
  AI_Pmaslo_sm_nizkoe_newHL := ai.Pmaslo_sm_nizkoe.dHL;
  AI_Pmaslo_sm_nizkoe_newLL := ai.Pmaslo_sm_nizkoe.dLL;
  AI_Pmaslo_sm_nizkoe_LW := ai.Pmaslo_sm_nizkoe.LW;
  AI_Pmaslo_sm_nizkoe_newLW := ai.Pmaslo_sm_nizkoe.dLW;
  AI_Pmaslo_sm_nizkoe_LA := ai.Pmaslo_sm_nizkoe.LA;
  AI_Pmaslo_sm_nizkoe_newLA := ai.Pmaslo_sm_nizkoe.dLA;

  AI_Pmaslo_sm_vysokoe_HL := ai.Pmaslo_sm_vysokoe.HL;
  AI_Pmaslo_sm_vysokoe_LL := ai.Pmaslo_sm_vysokoe.LL;
  AI_Pmaslo_sm_vysokoe_newHL := ai.Pmaslo_sm_vysokoe.dHL;
  AI_Pmaslo_sm_vysokoe_newLL := ai.Pmaslo_sm_vysokoe.dLL;
  AI_Pmaslo_sm_vysokoe_LW := ai.Pmaslo_sm_vysokoe.LW;
  AI_Pmaslo_sm_vysokoe_newLW := ai.Pmaslo_sm_vysokoe.dLW;
  AI_Pmaslo_sm_vysokoe_LA := ai.Pmaslo_sm_vysokoe.LA;
  AI_Pmaslo_sm_vysokoe_newLA := ai.Pmaslo_sm_vysokoe.dLA;

  AI_Pmasla_posle_GNS_HL := ai.Pmasla_posle_GNS.HL;
  AI_Pmasla_posle_GNS_LL := ai.Pmasla_posle_GNS.LL;
  AI_Pmasla_posle_GNS_newHL := ai.Pmasla_posle_GNS.dHL;
  AI_Pmasla_posle_GNS_newLL := ai.Pmasla_posle_GNS.dLL;
  AI_Pmasla_posle_GNS_HW := ai.Pmasla_posle_GNS.HW;
  AI_Pmasla_posle_GNS_newHW := ai.Pmasla_posle_GNS.dHW;
  AI_Pmasla_posle_GNS_LW := ai.Pmasla_posle_GNS.LW;
  AI_Pmasla_posle_GNS_newLW := ai.Pmasla_posle_GNS.dLW;

  AI_Pmasla_posle_NU_HL := ai.Pmasla_posle_NU.HL;
  AI_Pmasla_posle_NU_LL := ai.Pmasla_posle_NU.LL;
  AI_Pmasla_posle_NU_newHL := ai.Pmasla_posle_NU.dHL;
  AI_Pmasla_posle_NU_newLL := ai.Pmasla_posle_NU.dLL;
  AI_Pmasla_posle_NU_LW := ai.Pmasla_posle_NU.LW;
  AI_Pmasla_posle_NU_newLW := ai.Pmasla_posle_NU.dLW;

  AI_Pgaza_na_vhode_nagnetatelia_HL := ai.Pgaza_na_vhode_nagnetatelia.HL;
  AI_Pgaza_na_vhode_nagnetatelia_LL := ai.Pgaza_na_vhode_nagnetatelia.LL;
  AI_Pgaza_na_vhode_nagnetatelia_newHL := ai.Pgaza_na_vhode_nagnetatelia.dHL;
  AI_Pgaza_na_vhode_nagnetatelia_newLL := ai.Pgaza_na_vhode_nagnetatelia.dLL;
  AI_Pgaza_na_vhode_nagnetatelia_LW := ai.Pgaza_na_vhode_nagnetatelia.LW;
  AI_Pgaza_na_vhode_nagnetatelia_newLW := ai.Pgaza_na_vhode_nagnetatelia.dLW;

  AI_Pgaza_na_vyhode_nagnetatelia_HL := ai.Pgaza_na_vyhode_nagnetatelia.HL;
  AI_Pgaza_na_vyhode_nagnetatelia_LL := ai.Pgaza_na_vyhode_nagnetatelia.LL;
  AI_Pgaza_na_vyhode_nagnetatelia_newHL := ai.Pgaza_na_vyhode_nagnetatelia.dHL;
  AI_Pgaza_na_vyhode_nagnetatelia_newLL := ai.Pgaza_na_vyhode_nagnetatelia.dLL;
  AI_Pgaza_na_vyhode_nagnetatelia_LW := ai.Pgaza_na_vyhode_nagnetatelia.LW;
  AI_Pgaza_na_vyhode_nagnetatelia_newLW := ai.Pgaza_na_vyhode_nagnetatelia.dLW;
  AI_Pgaza_na_vyhode_nagnetatelia_HA := ai.Pgaza_na_vyhode_nagnetatelia.HA;
  AI_Pgaza_na_vyhode_nagnetatelia_newHA := ai.Pgaza_na_vyhode_nagnetatelia.dHA;

  AI_Pimpuls_gaz_HL := ai.Pimpuls_gaz.HL;
  AI_Pimpuls_gaz_LL := ai.Pimpuls_gaz.LL;
  AI_Pimpuls_gaz_newHL := ai.Pimpuls_gaz.dHL;
  AI_Pimpuls_gaz_newLL := ai.Pimpuls_gaz.dLL;
  AI_Pimpuls_gaz_LW := ai.Pimpuls_gaz.LW;
  AI_Pimpuls_gaz_newLW := ai.Pimpuls_gaz.dLW;

  AI_dPgaza_na_maslo_filtre_HL := ai.dPgaza_na_maslo_filtre.HL;
  AI_dPgaza_na_maslo_filtre_LL := ai.dPgaza_na_maslo_filtre.LL;
  AI_dPgaza_na_maslo_filtre_newHL := ai.dPgaza_na_maslo_filtre.dHL;
  AI_dPgaza_na_maslo_filtre_newLL := ai.dPgaza_na_maslo_filtre.dLL;
  AI_dPgaza_na_maslo_filtre_HW := ai.dPgaza_na_maslo_filtre.HW;
  AI_dPgaza_na_maslo_filtre_newHW := ai.dPgaza_na_maslo_filtre.dHW;

  AI_dPgaza_na_konfuzore_HL := ai.dPgaza_na_konfuzore.HL;
  AI_dPgaza_na_konfuzore_LL := ai.dPgaza_na_konfuzore.LL;
  AI_dPgaza_na_konfuzore_newHL := ai.dPgaza_na_konfuzore.dHL;
  AI_dPgaza_na_konfuzore_newLL := ai.dPgaza_na_konfuzore.dLL;
  AI_dPgaza_na_konfuzore_LW := ai.dPgaza_na_konfuzore.LW;
  AI_dPgaza_na_konfuzore_newLW := ai.dPgaza_na_konfuzore.dLW;

  AI_dPmaslo_gaz_HL := ai.dPmaslo_gaz.HL;
  AI_dPmaslo_gaz_LL := ai.dPmaslo_gaz.LL;
  AI_dPmaslo_gaz_newHL := ai.dPmaslo_gaz.dHL;
  AI_dPmaslo_gaz_newLL := ai.dPmaslo_gaz.dLL;
  AI_dPmaslo_gaz_LW := ai.dPmaslo_gaz.LW;
  AI_dPmaslo_gaz_newLW := ai.dPmaslo_gaz.dLW;
  AI_dPmaslo_gaz_LA := ai.dPmaslo_gaz.LA;
  AI_dPmaslo_gaz_newLA := ai.dPmaslo_gaz.dLA;

  AI_Os_sdvig_nagnetatelja_plus_HL := ai.Os_sdvig_nagnetatelja_plus.HL;
  AI_Os_sdvig_nagnetatelja_plus_LL := ai.Os_sdvig_nagnetatelja_plus.LL;
  AI_Os_sdvig_nagnetatelja_plus_newHL := ai.Os_sdvig_nagnetatelja_plus.dHL;
  AI_Os_sdvig_nagnetatelja_plus_newLL := ai.Os_sdvig_nagnetatelja_plus.dLL;
  AI_Os_sdvig_nagnetatelja_plus_HW := ai.Os_sdvig_nagnetatelja_plus.HW;
  AI_Os_sdvig_nagnetatelja_plus_newHW := ai.Os_sdvig_nagnetatelja_plus.dHW;
  AI_Os_sdvig_nagnetatelja_plus_HA := ai.Os_sdvig_nagnetatelja_plus.HA;
  AI_Os_sdvig_nagnetatelja_plus_newHA := ai.Os_sdvig_nagnetatelja_plus.dHA;

  AI_Os_sdvig_nagnetatelja_minus_HL := ai.Os_sdvig_nagnetatelja_minus.HL;
  AI_Os_sdvig_nagnetatelja_minus_LL := ai.Os_sdvig_nagnetatelja_minus.LL;
  AI_Os_sdvig_nagnetatelja_minus_newHL := ai.Os_sdvig_nagnetatelja_minus.dHL;
  AI_Os_sdvig_nagnetatelja_minus_newLL := ai.Os_sdvig_nagnetatelja_minus.dLL;
  AI_Os_sdvig_nagnetatelja_minus_LW := ai.Os_sdvig_nagnetatelja_minus.LW;
  AI_Os_sdvig_nagnetatelja_minus_newLW := ai.Os_sdvig_nagnetatelja_minus.dLW;
  AI_Os_sdvig_nagnetatelja_minus_LA := ai.Os_sdvig_nagnetatelja_minus.LA;
  AI_Os_sdvig_nagnetatelja_minus_newLA := ai.Os_sdvig_nagnetatelja_minus.dLA;

  AI_Yroven_masla_MB_HL := ai.Yroven_masla_MB.HL;
  AI_Yroven_masla_MB_LL := ai.Yroven_masla_MB.LL;
  AI_Yroven_masla_MB_newHL := ai.Yroven_masla_MB.dHL;
  AI_Yroven_masla_MB_newLL := ai.Yroven_masla_MB.dLL;
  AI_Yroven_masla_MB_LW := ai.Yroven_masla_MB.LW;
  AI_Yroven_masla_MB_newLW := ai.Yroven_masla_MB.dLW;

  AI_Kontrol_per_220V_HL := ai.Kontrol_per_220V.HL;
  AI_Kontrol_per_220V_LL := ai.Kontrol_per_220V.LL;
  AI_Kontrol_per_220V_newHL := ai.Kontrol_per_220V.dHL;
  AI_Kontrol_per_220V_newLL := ai.Kontrol_per_220V.dLL;
  AI_Kontrol_per_220V_HW := ai.Kontrol_per_220V.HW;
  AI_Kontrol_per_220V_newHW := ai.Kontrol_per_220V.dHW;
  AI_Kontrol_per_220V_LW := ai.Kontrol_per_220V.LW;
  AI_Kontrol_per_220V_newLW := ai.Kontrol_per_220V.dLW;

  AI_Kontrol_post_220V_HL := ai.Kontrol_post_220V.HL;
  AI_Kontrol_post_220V_LL := ai.Kontrol_post_220V.LL;
  AI_Kontrol_post_220V_newHL := ai.Kontrol_post_220V.dHL;
  AI_Kontrol_post_220V_newLL := ai.Kontrol_post_220V.dLL;
  AI_Kontrol_post_220V_HW := ai.Kontrol_post_220V.HW;
  AI_Kontrol_post_220V_newHW := ai.Kontrol_post_220V.dHW;
  AI_Kontrol_post_220V_LW := ai.Kontrol_post_220V.LW;
  AI_Kontrol_post_220V_newLW := ai.Kontrol_post_220V.dLW;

  AI_Tok_statora_HL := ai.Tok_statora.HL;
  AI_Tok_statora_LL := ai.Tok_statora.LL;
  AI_Tok_statora_newHL := ai.Tok_statora.dHL;
  AI_Tok_statora_newLL := ai.Tok_statora.dLL;
  AI_Tok_statora_LW := ai.Tok_statora.LW;
  AI_Tok_statora_newLW := ai.Tok_statora.dLW;

  AI_Vibro_skorost_OPED_T1_HL := ai.Vibro_skorost_OPED_T1.HL;
  AI_Vibro_skorost_OPED_T1_LL := ai.Vibro_skorost_OPED_T1.LL;
  AI_Vibro_skorost_OPED_T1_newHL := ai.Vibro_skorost_OPED_T1.dHL;
  AI_Vibro_skorost_OPED_T1_newLL := ai.Vibro_skorost_OPED_T1.dLL;
  AI_Vibro_skorost_OPED_T1_HW := ai.Vibro_skorost_OPED_T1.HW;
  AI_Vibro_skorost_OPED_T1_newHW := ai.Vibro_skorost_OPED_T1.dHW;
  AI_Vibro_skorost_OPED_T1_HA := ai.Vibro_skorost_OPED_T1.HA;
  AI_Vibro_skorost_OPED_T1_newHA := ai.Vibro_skorost_OPED_T1.dHA;

  AI_Vibro_skorost_OYPED_T2_HL := ai.Vibro_skorost_OYPED_T2.HL;
  AI_Vibro_skorost_OYPED_T2_LL := ai.Vibro_skorost_OYPED_T2.LL;
  AI_Vibro_skorost_OYPED_T2_newHL := ai.Vibro_skorost_OYPED_T2.dHL;
  AI_Vibro_skorost_OYPED_T2_newLL := ai.Vibro_skorost_OYPED_T2.dLL;
  AI_Vibro_skorost_OYPED_T2_HW := ai.Vibro_skorost_OYPED_T2.HW;
  AI_Vibro_skorost_OYPED_T2_newHW := ai.Vibro_skorost_OYPED_T2.dHW;
  AI_Vibro_skorost_OYPED_T2_HA := ai.Vibro_skorost_OYPED_T2.HA;
  AI_Vibro_skorost_OYPED_T2_newHA := ai.Vibro_skorost_OYPED_T2.dHA;

  AI_Vibro_skorost_OYP_kolesa_ED_T3_HL := ai.Vibro_skorost_OYP_kolesa_ED_T3.HL;
  AI_Vibro_skorost_OYP_kolesa_ED_T3_LL := ai.Vibro_skorost_OYP_kolesa_ED_T3.LL;
  AI_Vibro_skorost_OYP_kolesa_ED_T3_newHL := ai.Vibro_skorost_OYP_kolesa_ED_T3.dHL;
  AI_Vibro_skorost_OYP_kolesa_ED_T3_newLL := ai.Vibro_skorost_OYP_kolesa_ED_T3.dLL;
  AI_Vibro_skorost_OYP_kolesa_ED_T3_HW := ai.Vibro_skorost_OYP_kolesa_ED_T3.HW;
  AI_Vibro_skorost_OYP_kolesa_ED_T3_newHW := ai.Vibro_skorost_OYP_kolesa_ED_T3.dHW;
  AI_Vibro_skorost_OYP_kolesa_ED_T3_HA := ai.Vibro_skorost_OYP_kolesa_ED_T3.HA;
  AI_Vibro_skorost_OYP_kolesa_ED_T3_newHA := ai.Vibro_skorost_OYP_kolesa_ED_T3.dHA;

  AI_Vibro_skorost_OP_kolesa_RH_T4_HL := ai.Vibro_skorost_OP_kolesa_RH_T4.HL;
  AI_Vibro_skorost_OP_kolesa_RH_T4_LL := ai.Vibro_skorost_OP_kolesa_RH_T4.LL;
  AI_Vibro_skorost_OP_kolesa_RH_T4_newHL := ai.Vibro_skorost_OP_kolesa_RH_T4.dHL;
  AI_Vibro_skorost_OP_kolesa_RH_T4_newLL := ai.Vibro_skorost_OP_kolesa_RH_T4.dLL;
  AI_Vibro_skorost_OP_kolesa_RH_T4_HW := ai.Vibro_skorost_OP_kolesa_RH_T4.HW;
  AI_Vibro_skorost_OP_kolesa_RH_T4_newHW := ai.Vibro_skorost_OP_kolesa_RH_T4.dHW;
  AI_Vibro_skorost_OP_kolesa_RH_T4_HA := ai.Vibro_skorost_OP_kolesa_RH_T4.HA;
  AI_Vibro_skorost_OP_kolesa_RH_T4_newHA := ai.Vibro_skorost_OP_kolesa_RH_T4.dHA;

  AI_Vibro_skorost_OP_shesterni_RED_T5_HL := ai.Vibro_skorost_OP_shesterni_RED_T5.HL;
  AI_Vibro_skorost_OP_shesterni_RED_T5_LL := ai.Vibro_skorost_OP_shesterni_RED_T5.LL;
  AI_Vibro_skorost_OP_shesterni_RED_T5_newHL := ai.Vibro_skorost_OP_shesterni_RED_T5.dHL;
  AI_Vibro_skorost_OP_shesterni_RED_T5_newLL := ai.Vibro_skorost_OP_shesterni_RED_T5.dLL;
  AI_Vibro_skorost_OP_shesterni_RED_T5_HW := ai.Vibro_skorost_OP_shesterni_RED_T5.HW;
  AI_Vibro_skorost_OP_shesterni_RED_T5_newHW := ai.Vibro_skorost_OP_shesterni_RED_T5.dHW;
  AI_Vibro_skorost_OP_shesterni_RED_T5_HA := ai.Vibro_skorost_OP_shesterni_RED_T5.HA;
  AI_Vibro_skorost_OP_shesterni_RED_T5_newHA := ai.Vibro_skorost_OP_shesterni_RED_T5.dHA;

  AI_Vibro_skorost_OP_shesterni_RED_T6_HL := ai.Vibro_skorost_OP_shesterni_RED_T6.HL;
  AI_Vibro_skorost_OP_shesterni_RED_T6_LL := ai.Vibro_skorost_OP_shesterni_RED_T6.LL;
  AI_Vibro_skorost_OP_shesterni_RED_T6_newHL := ai.Vibro_skorost_OP_shesterni_RED_T6.dHL;
  AI_Vibro_skorost_OP_shesterni_RED_T6_newLL := ai.Vibro_skorost_OP_shesterni_RED_T6.dLL;
  AI_Vibro_skorost_OP_shesterni_RED_T6_HW := ai.Vibro_skorost_OP_shesterni_RED_T6.HW;
  AI_Vibro_skorost_OP_shesterni_RED_T6_newHW := ai.Vibro_skorost_OP_shesterni_RED_T6.dHW;
  AI_Vibro_skorost_OP_shesterni_RED_T6_HA := ai.Vibro_skorost_OP_shesterni_RED_T6.HA;
  AI_Vibro_skorost_OP_shesterni_RED_T6_newHA := ai.Vibro_skorost_OP_shesterni_RED_T6.dHA;
END_FUNCTION_BLOCK

FUNCTION_BLOCK OPC_AI_GET
  VAR_EXTERNAL
    ai : aiConfig;
    AI_Tstali_statora_kanal_1_HL : LREAL;
    AI_Tstali_statora_kanal_1_LL : LREAL;
    AI_Tstali_statora_kanal_1_command : UINT;
    AI_Tstali_statora_kanal_1_newHL : LREAL;
    AI_Tstali_statora_kanal_1_newLL : LREAL;
    AI_Tstali_statora_kanal_1_status : UDINT;
    AI_Tstali_statora_kanal_1_value : LREAL;
    AI_Tstali_statora_kanal_1_HW : LREAL;
    AI_Tstali_statora_kanal_1_newHW : LREAL;
    AI_Tstali_statora_kanal_2_HL : LREAL;
    AI_Tstali_statora_kanal_2_LL : LREAL;
    AI_Tstali_statora_kanal_2_command : UINT;
    AI_Tstali_statora_kanal_2_newHL : LREAL;
    AI_Tstali_statora_kanal_2_newLL : LREAL;
    AI_Tstali_statora_kanal_2_status : UDINT;
    AI_Tstali_statora_kanal_2_value : LREAL;
    AI_Tstali_statora_kanal_2_HW : LREAL;
    AI_Tstali_statora_kanal_2_newHW : LREAL;
    AI_Tstali_statora_kanal_3_HL : LREAL;
    AI_Tstali_statora_kanal_3_LL : LREAL;
    AI_Tstali_statora_kanal_3_command : UINT;
    AI_Tstali_statora_kanal_3_newHL : LREAL;
    AI_Tstali_statora_kanal_3_newLL : LREAL;
    AI_Tstali_statora_kanal_3_status : UDINT;
    AI_Tstali_statora_kanal_3_value : LREAL;
    AI_Tstali_statora_kanal_3_HW : LREAL;
    AI_Tstali_statora_kanal_3_newHW : LREAL;
    AI_Tmedi_statora_kanal_1_HL : LREAL;
    AI_Tmedi_statora_kanal_1_LL : LREAL;
    AI_Tmedi_statora_kanal_1_command : UINT;
    AI_Tmedi_statora_kanal_1_newHL : LREAL;
    AI_Tmedi_statora_kanal_1_newLL : LREAL;
    AI_Tmedi_statora_kanal_1_status : UDINT;
    AI_Tmedi_statora_kanal_1_value : LREAL;
    AI_Tmedi_statora_kanal_1_HW : LREAL;
    AI_Tmedi_statora_kanal_1_newHW : LREAL;
    AI_Tmedi_statora_kanal_2_HL : LREAL;
    AI_Tmedi_statora_kanal_2_LL : LREAL;
    AI_Tmedi_statora_kanal_2_command : UINT;
    AI_Tmedi_statora_kanal_2_newHL : LREAL;
    AI_Tmedi_statora_kanal_2_newLL : LREAL;
    AI_Tmedi_statora_kanal_2_status : UDINT;
    AI_Tmedi_statora_kanal_2_value : LREAL;
    AI_Tmedi_statora_kanal_2_HW : LREAL;
    AI_Tmedi_statora_kanal_2_newHW : LREAL;
    AI_Tmedi_statora_kanal_3_HL : LREAL;
    AI_Tmedi_statora_kanal_3_LL : LREAL;
    AI_Tmedi_statora_kanal_3_command : UINT;
    AI_Tmedi_statora_kanal_3_newHL : LREAL;
    AI_Tmedi_statora_kanal_3_newLL : LREAL;
    AI_Tmedi_statora_kanal_3_status : UDINT;
    AI_Tmedi_statora_kanal_3_value : LREAL;
    AI_Tmedi_statora_kanal_3_HW : LREAL;
    AI_Tmedi_statora_kanal_3_newHW : LREAL;
    AI_Toporno_podshipnika_EDT_1_HL : LREAL;
    AI_Toporno_podshipnika_EDT_1_LL : LREAL;
    AI_Toporno_podshipnika_EDT_1_command : UINT;
    AI_Toporno_podshipnika_EDT_1_newHL : LREAL;
    AI_Toporno_podshipnika_EDT_1_newLL : LREAL;
    AI_Toporno_podshipnika_EDT_1_status : UDINT;
    AI_Toporno_podshipnika_EDT_1_value : LREAL;
    AI_Toporno_podshipnika_EDT_1_HW : LREAL;
    AI_Toporno_podshipnika_EDT_1_newHW : LREAL;
    AI_Toporno_podshipnika_EDT_1_HA : LREAL;
    AI_Toporno_podshipnika_EDT_1_newHA : LREAL;
    AI_Toy_podshipnika_EDT_2_HL : LREAL;
    AI_Toy_podshipnika_EDT_2_LL : LREAL;
    AI_Toy_podshipnika_EDT_2_command : UINT;
    AI_Toy_podshipnika_EDT_2_newHL : LREAL;
    AI_Toy_podshipnika_EDT_2_newLL : LREAL;
    AI_Toy_podshipnika_EDT_2_status : UDINT;
    AI_Toy_podshipnika_EDT_2_value : LREAL;
    AI_Toy_podshipnika_EDT_2_HW : LREAL;
    AI_Toy_podshipnika_EDT_2_newHW : LREAL;
    AI_Toy_podshipnika_EDT_2_HA : LREAL;
    AI_Toy_podshipnika_EDT_2_newHA : LREAL;
    AI_Toy_podshipnika_kol_EDT_3_HL : LREAL;
    AI_Toy_podshipnika_kol_EDT_3_LL : LREAL;
    AI_Toy_podshipnika_kol_EDT_3_command : UINT;
    AI_Toy_podshipnika_kol_EDT_3_newHL : LREAL;
    AI_Toy_podshipnika_kol_EDT_3_newLL : LREAL;
    AI_Toy_podshipnika_kol_EDT_3_status : UDINT;
    AI_Toy_podshipnika_kol_EDT_3_value : LREAL;
    AI_Toy_podshipnika_kol_EDT_3_HW : LREAL;
    AI_Toy_podshipnika_kol_EDT_3_newHW : LREAL;
    AI_Toy_podshipnika_kol_EDT_3_HA : LREAL;
    AI_Toy_podshipnika_kol_EDT_3_newHA : LREAL;
    AI_Toy_podshipnika_kol_EDT_4_HL : LREAL;
    AI_Toy_podshipnika_kol_EDT_4_LL : LREAL;
    AI_Toy_podshipnika_kol_EDT_4_command : UINT;
    AI_Toy_podshipnika_kol_EDT_4_newHL : LREAL;
    AI_Toy_podshipnika_kol_EDT_4_newLL : LREAL;
    AI_Toy_podshipnika_kol_EDT_4_status : UDINT;
    AI_Toy_podshipnika_kol_EDT_4_value : LREAL;
    AI_Toy_podshipnika_kol_EDT_4_HW : LREAL;
    AI_Toy_podshipnika_kol_EDT_4_newHW : LREAL;
    AI_Toy_podshipnika_kol_EDT_4_HA : LREAL;
    AI_Toy_podshipnika_kol_EDT_4_newHA : LREAL;
    AI_Toy_podshipnika_shest_red_EDT_5_HL : LREAL;
    AI_Toy_podshipnika_shest_red_EDT_5_LL : LREAL;
    AI_Toy_podshipnika_shest_red_EDT_5_command : UINT;
    AI_Toy_podshipnika_shest_red_EDT_5_newHL : LREAL;
    AI_Toy_podshipnika_shest_red_EDT_5_newLL : LREAL;
    AI_Toy_podshipnika_shest_red_EDT_5_status : UDINT;
    AI_Toy_podshipnika_shest_red_EDT_5_value : LREAL;
    AI_Toy_podshipnika_shest_red_EDT_5_HW : LREAL;
    AI_Toy_podshipnika_shest_red_EDT_5_newHW : LREAL;
    AI_Toy_podshipnika_shest_red_EDT_5_HA : LREAL;
    AI_Toy_podshipnika_shest_red_EDT_5_newHA : LREAL;
    AI_Ty_podshipnika_red_EDT_6_HL : LREAL;
    AI_Ty_podshipnika_red_EDT_6_LL : LREAL;
    AI_Ty_podshipnika_red_EDT_6_command : UINT;
    AI_Ty_podshipnika_red_EDT_6_newHL : LREAL;
    AI_Ty_podshipnika_red_EDT_6_newLL : LREAL;
    AI_Ty_podshipnika_red_EDT_6_status : UDINT;
    AI_Ty_podshipnika_red_EDT_6_value : LREAL;
    AI_Ty_podshipnika_red_EDT_6_HW : LREAL;
    AI_Ty_podshipnika_red_EDT_6_newHW : LREAL;
    AI_Ty_podshipnika_red_EDT_6_HA : LREAL;
    AI_Ty_podshipnika_red_EDT_6_newHA : LREAL;
    AI_Ty_podshipnika_nagnet_EDT_7_1_HL : LREAL;
    AI_Ty_podshipnika_nagnet_EDT_7_1_LL : LREAL;
    AI_Ty_podshipnika_nagnet_EDT_7_1_command : UINT;
    AI_Ty_podshipnika_nagnet_EDT_7_1_newHL : LREAL;
    AI_Ty_podshipnika_nagnet_EDT_7_1_newLL : LREAL;
    AI_Ty_podshipnika_nagnet_EDT_7_1_status : UDINT;
    AI_Ty_podshipnika_nagnet_EDT_7_1_value : LREAL;
    AI_Ty_podshipnika_nagnet_EDT_7_1_HW : LREAL;
    AI_Ty_podshipnika_nagnet_EDT_7_1_newHW : LREAL;
    AI_Ty_podshipnika_nagnet_EDT_7_1_HA : LREAL;
    AI_Ty_podshipnika_nagnet_EDT_7_1_newHA : LREAL;
    AI_Ty_podshipnika_nagnet_EDT_7_2_HL : LREAL;
    AI_Ty_podshipnika_nagnet_EDT_7_2_LL : LREAL;
    AI_Ty_podshipnika_nagnet_EDT_7_2_command : UINT;
    AI_Ty_podshipnika_nagnet_EDT_7_2_newHL : LREAL;
    AI_Ty_podshipnika_nagnet_EDT_7_2_newLL : LREAL;
    AI_Ty_podshipnika_nagnet_EDT_7_2_status : UDINT;
    AI_Ty_podshipnika_nagnet_EDT_7_2_value : LREAL;
    AI_Ty_podshipnika_nagnet_EDT_7_2_HW : LREAL;
    AI_Ty_podshipnika_nagnet_EDT_7_2_newHW : LREAL;
    AI_Ty_podshipnika_nagnet_EDT_7_2_HA : LREAL;
    AI_Ty_podshipnika_nagnet_EDT_7_2_newHA : LREAL;
    AI_Toy_podshipnika_svobod_konca_EDT_8_1_HL : LREAL;
    AI_Toy_podshipnika_svobod_konca_EDT_8_1_LL : LREAL;
    AI_Toy_podshipnika_svobod_konca_EDT_8_1_command : UINT;
    AI_Toy_podshipnika_svobod_konca_EDT_8_1_newHL : LREAL;
    AI_Toy_podshipnika_svobod_konca_EDT_8_1_newLL : LREAL;
    AI_Toy_podshipnika_svobod_konca_EDT_8_1_status : UDINT;
    AI_Toy_podshipnika_svobod_konca_EDT_8_1_value : LREAL;
    AI_Toy_podshipnika_svobod_konca_EDT_8_1_HW : LREAL;
    AI_Toy_podshipnika_svobod_konca_EDT_8_1_newHW : LREAL;
    AI_Toy_podshipnika_svobod_konca_EDT_8_1_HA : LREAL;
    AI_Toy_podshipnika_svobod_konca_EDT_8_1_newHA : LREAL;
    AI_Toy_podshipnika_svobod_konca_EDT_8_2_HL : LREAL;
    AI_Toy_podshipnika_svobod_konca_EDT_8_2_LL : LREAL;
    AI_Toy_podshipnika_svobod_konca_EDT_8_2_command : UINT;
    AI_Toy_podshipnika_svobod_konca_EDT_8_2_newHL : LREAL;
    AI_Toy_podshipnika_svobod_konca_EDT_8_2_newLL : LREAL;
    AI_Toy_podshipnika_svobod_konca_EDT_8_2_status : UDINT;
    AI_Toy_podshipnika_svobod_konca_EDT_8_2_value : LREAL;
    AI_Toy_podshipnika_svobod_konca_EDT_8_2_HW : LREAL;
    AI_Toy_podshipnika_svobod_konca_EDT_8_2_newHW : LREAL;
    AI_Toy_podshipnika_svobod_konca_EDT_8_2_HA : LREAL;
    AI_Toy_podshipnika_svobod_konca_EDT_8_2_newHA : LREAL;
    AI_Toy_podshipnika_rab_kol_EDT_9_1_HL : LREAL;
    AI_Toy_podshipnika_rab_kol_EDT_9_1_LL : LREAL;
    AI_Toy_podshipnika_rab_kol_EDT_9_1_command : UINT;
    AI_Toy_podshipnika_rab_kol_EDT_9_1_newHL : LREAL;
    AI_Toy_podshipnika_rab_kol_EDT_9_1_newLL : LREAL;
    AI_Toy_podshipnika_rab_kol_EDT_9_1_status : UDINT;
    AI_Toy_podshipnika_rab_kol_EDT_9_1_value : LREAL;
    AI_Toy_podshipnika_rab_kol_EDT_9_1_HW : LREAL;
    AI_Toy_podshipnika_rab_kol_EDT_9_1_newHW : LREAL;
    AI_Toy_podshipnika_rab_kol_EDT_9_1_HA : LREAL;
    AI_Toy_podshipnika_rab_kol_EDT_9_1_newHA : LREAL;
    AI_Toy_podshipnika_rab_kol_EDT_9_2_HL : LREAL;
    AI_Toy_podshipnika_rab_kol_EDT_9_2_LL : LREAL;
    AI_Toy_podshipnika_rab_kol_EDT_9_2_command : UINT;
    AI_Toy_podshipnika_rab_kol_EDT_9_2_newHL : LREAL;
    AI_Toy_podshipnika_rab_kol_EDT_9_2_newLL : LREAL;
    AI_Toy_podshipnika_rab_kol_EDT_9_2_status : UDINT;
    AI_Toy_podshipnika_rab_kol_EDT_9_2_value : LREAL;
    AI_Toy_podshipnika_rab_kol_EDT_9_2_HW : LREAL;
    AI_Toy_podshipnika_rab_kol_EDT_9_2_newHW : LREAL;
    AI_Toy_podshipnika_rab_kol_EDT_9_2_HA : LREAL;
    AI_Toy_podshipnika_rab_kol_EDT_9_2_newHA : LREAL;
    AI_Toy_podshipnika_nerab_kol_EDT_10_1_HL : LREAL;
    AI_Toy_podshipnika_nerab_kol_EDT_10_1_LL : LREAL;
    AI_Toy_podshipnika_nerab_kol_EDT_10_1_command : UINT;
    AI_Toy_podshipnika_nerab_kol_EDT_10_1_newHL : LREAL;
    AI_Toy_podshipnika_nerab_kol_EDT_10_1_newLL : LREAL;
    AI_Toy_podshipnika_nerab_kol_EDT_10_1_status : UDINT;
    AI_Toy_podshipnika_nerab_kol_EDT_10_1_value : LREAL;
    AI_Toy_podshipnika_nerab_kol_EDT_10_1_HW : LREAL;
    AI_Toy_podshipnika_nerab_kol_EDT_10_1_newHW : LREAL;
    AI_Toy_podshipnika_nerab_kol_EDT_10_1_HA : LREAL;
    AI_Toy_podshipnika_nerab_kol_EDT_10_1_newHA : LREAL;
    AI_Toy_podshipnika_nerab_kol_EDT_10_2_HL : LREAL;
    AI_Toy_podshipnika_nerab_kol_EDT_10_2_LL : LREAL;
    AI_Toy_podshipnika_nerab_kol_EDT_10_2_command : UINT;
    AI_Toy_podshipnika_nerab_kol_EDT_10_2_newHL : LREAL;
    AI_Toy_podshipnika_nerab_kol_EDT_10_2_newLL : LREAL;
    AI_Toy_podshipnika_nerab_kol_EDT_10_2_status : UDINT;
    AI_Toy_podshipnika_nerab_kol_EDT_10_2_value : LREAL;
    AI_Toy_podshipnika_nerab_kol_EDT_10_2_HW : LREAL;
    AI_Toy_podshipnika_nerab_kol_EDT_10_2_newHW : LREAL;
    AI_Toy_podshipnika_nerab_kol_EDT_10_2_HA : LREAL;
    AI_Toy_podshipnika_nerab_kol_EDT_10_2_newHA : LREAL;
    AI_Tholodnogo_vozduha_ED_kanal_1_HL : LREAL;
    AI_Tholodnogo_vozduha_ED_kanal_1_LL : LREAL;
    AI_Tholodnogo_vozduha_ED_kanal_1_command : UINT;
    AI_Tholodnogo_vozduha_ED_kanal_1_newHL : LREAL;
    AI_Tholodnogo_vozduha_ED_kanal_1_newLL : LREAL;
    AI_Tholodnogo_vozduha_ED_kanal_1_status : UDINT;
    AI_Tholodnogo_vozduha_ED_kanal_1_value : LREAL;
    AI_Tholodnogo_vozduha_ED_kanal_1_HW : LREAL;
    AI_Tholodnogo_vozduha_ED_kanal_1_newHW : LREAL;
    AI_Tholodnogo_vozduha_ED_kanal_2_HL : LREAL;
    AI_Tholodnogo_vozduha_ED_kanal_2_LL : LREAL;
    AI_Tholodnogo_vozduha_ED_kanal_2_command : UINT;
    AI_Tholodnogo_vozduha_ED_kanal_2_newHL : LREAL;
    AI_Tholodnogo_vozduha_ED_kanal_2_newLL : LREAL;
    AI_Tholodnogo_vozduha_ED_kanal_2_status : UDINT;
    AI_Tholodnogo_vozduha_ED_kanal_2_value : LREAL;
    AI_Tholodnogo_vozduha_ED_kanal_2_HW : LREAL;
    AI_Tholodnogo_vozduha_ED_kanal_2_newHW : LREAL;
    AI_Tgorjachego_vozduha_ED_kanal_1_HL : LREAL;
    AI_Tgorjachego_vozduha_ED_kanal_1_LL : LREAL;
    AI_Tgorjachego_vozduha_ED_kanal_1_command : UINT;
    AI_Tgorjachego_vozduha_ED_kanal_1_newHL : LREAL;
    AI_Tgorjachego_vozduha_ED_kanal_1_newLL : LREAL;
    AI_Tgorjachego_vozduha_ED_kanal_1_status : UDINT;
    AI_Tgorjachego_vozduha_ED_kanal_1_value : LREAL;
    AI_Tgorjachego_vozduha_ED_kanal_1_HW : LREAL;
    AI_Tgorjachego_vozduha_ED_kanal_1_newHW : LREAL;
    AI_Tgorjachego_vozduha_ED_kanal_2_HL : LREAL;
    AI_Tgorjachego_vozduha_ED_kanal_2_LL : LREAL;
    AI_Tgorjachego_vozduha_ED_kanal_2_command : UINT;
    AI_Tgorjachego_vozduha_ED_kanal_2_newHL : LREAL;
    AI_Tgorjachego_vozduha_ED_kanal_2_newLL : LREAL;
    AI_Tgorjachego_vozduha_ED_kanal_2_status : UDINT;
    AI_Tgorjachego_vozduha_ED_kanal_2_value : LREAL;
    AI_Tgorjachego_vozduha_ED_kanal_2_HW : LREAL;
    AI_Tgorjachego_vozduha_ED_kanal_2_newHW : LREAL;
    AI_Tnarujnogo_vozduha_HL : LREAL;
    AI_Tnarujnogo_vozduha_LL : LREAL;
    AI_Tnarujnogo_vozduha_command : UINT;
    AI_Tnarujnogo_vozduha_newHL : LREAL;
    AI_Tnarujnogo_vozduha_newLL : LREAL;
    AI_Tnarujnogo_vozduha_status : UDINT;
    AI_Tnarujnogo_vozduha_value : LREAL;
    AI_Tnarujnogo_vozduha_HW : LREAL;
    AI_Tnarujnogo_vozduha_newHW : LREAL;
    AI_Tgaza_na_vhode_H_HL : LREAL;
    AI_Tgaza_na_vhode_H_LL : LREAL;
    AI_Tgaza_na_vhode_H_command : UINT;
    AI_Tgaza_na_vhode_H_newHL : LREAL;
    AI_Tgaza_na_vhode_H_newLL : LREAL;
    AI_Tgaza_na_vhode_H_status : UDINT;
    AI_Tgaza_na_vhode_H_value : LREAL;
    AI_Tgaza_na_vhode_H_HW : LREAL;
    AI_Tgaza_na_vhode_H_newHW : LREAL;
    AI_Tgaza_na_vyhode_H_HL : LREAL;
    AI_Tgaza_na_vyhode_H_LL : LREAL;
    AI_Tgaza_na_vyhode_H_command : UINT;
    AI_Tgaza_na_vyhode_H_newHL : LREAL;
    AI_Tgaza_na_vyhode_H_newLL : LREAL;
    AI_Tgaza_na_vyhode_H_status : UDINT;
    AI_Tgaza_na_vyhode_H_value : LREAL;
    AI_Tgaza_na_vyhode_H_HW : LREAL;
    AI_Tgaza_na_vyhode_H_newHW : LREAL;
    AI_Tgaza_na_vyhode_H_HA : LREAL;
    AI_Tgaza_na_vyhode_H_newHA : LREAL;
    AI_Tmasla_do_AVOM_HL : LREAL;
    AI_Tmasla_do_AVOM_LL : LREAL;
    AI_Tmasla_do_AVOM_command : UINT;
    AI_Tmasla_do_AVOM_newHL : LREAL;
    AI_Tmasla_do_AVOM_newLL : LREAL;
    AI_Tmasla_do_AVOM_status : UDINT;
    AI_Tmasla_do_AVOM_value : LREAL;
    AI_Tmasla_do_AVOM_HW : LREAL;
    AI_Tmasla_do_AVOM_newHW : LREAL;
    AI_Tmasla_posle_AVOM_HL : LREAL;
    AI_Tmasla_posle_AVOM_LL : LREAL;
    AI_Tmasla_posle_AVOM_command : UINT;
    AI_Tmasla_posle_AVOM_newHL : LREAL;
    AI_Tmasla_posle_AVOM_newLL : LREAL;
    AI_Tmasla_posle_AVOM_status : UDINT;
    AI_Tmasla_posle_AVOM_value : LREAL;
    AI_Tmasla_posle_AVOM_HW : LREAL;
    AI_Tmasla_posle_AVOM_newHW : LREAL;
    AI_Tmasla_MB_HL : LREAL;
    AI_Tmasla_MB_LL : LREAL;
    AI_Tmasla_MB_command : UINT;
    AI_Tmasla_MB_newHL : LREAL;
    AI_Tmasla_MB_newLL : LREAL;
    AI_Tmasla_MB_status : UDINT;
    AI_Tmasla_MB_value : LREAL;
    AI_Tmasla_MB_HW : LREAL;
    AI_Tmasla_MB_newHW : LREAL;
    AI_Tmasla_MB_TEN_HL : LREAL;
    AI_Tmasla_MB_TEN_LL : LREAL;
    AI_Tmasla_MB_TEN_command : UINT;
    AI_Tmasla_MB_TEN_newHL : LREAL;
    AI_Tmasla_MB_TEN_newLL : LREAL;
    AI_Tmasla_MB_TEN_status : UDINT;
    AI_Tmasla_MB_TEN_value : LREAL;
    AI_Tmasla_MB_TEN_HW : LREAL;
    AI_Tmasla_MB_TEN_newHW : LREAL;
    AI_Tshu_HL : LREAL;
    AI_Tshu_LL : LREAL;
    AI_Tshu_command : UINT;
    AI_Tshu_newHL : LREAL;
    AI_Tshu_newLL : LREAL;
    AI_Tshu_status : UDINT;
    AI_Tshu_value : LREAL;
    AI_Pmaslo_sm_nizkoe_HL : LREAL;
    AI_Pmaslo_sm_nizkoe_LL : LREAL;
    AI_Pmaslo_sm_nizkoe_command : UINT;
    AI_Pmaslo_sm_nizkoe_newHL : LREAL;
    AI_Pmaslo_sm_nizkoe_newLL : LREAL;
    AI_Pmaslo_sm_nizkoe_status : UDINT;
    AI_Pmaslo_sm_nizkoe_value : LREAL;
    AI_Pmaslo_sm_nizkoe_LW : LREAL;
    AI_Pmaslo_sm_nizkoe_newLW : LREAL;
    AI_Pmaslo_sm_nizkoe_LA : LREAL;
    AI_Pmaslo_sm_nizkoe_newLA : LREAL;
    AI_Pmaslo_sm_vysokoe_HL : LREAL;
    AI_Pmaslo_sm_vysokoe_LL : LREAL;
    AI_Pmaslo_sm_vysokoe_command : UINT;
    AI_Pmaslo_sm_vysokoe_newHL : LREAL;
    AI_Pmaslo_sm_vysokoe_newLL : LREAL;
    AI_Pmaslo_sm_vysokoe_status : UDINT;
    AI_Pmaslo_sm_vysokoe_value : LREAL;
    AI_Pmaslo_sm_vysokoe_LW : LREAL;
    AI_Pmaslo_sm_vysokoe_newLW : LREAL;
    AI_Pmaslo_sm_vysokoe_LA : LREAL;
    AI_Pmaslo_sm_vysokoe_newLA : LREAL;
    AI_Pmasla_posle_GNS_HL : LREAL;
    AI_Pmasla_posle_GNS_LL : LREAL;
    AI_Pmasla_posle_GNS_command : UINT;
    AI_Pmasla_posle_GNS_newHL : LREAL;
    AI_Pmasla_posle_GNS_newLL : LREAL;
    AI_Pmasla_posle_GNS_status : UDINT;
    AI_Pmasla_posle_GNS_value : LREAL;
    AI_Pmasla_posle_GNS_HW : LREAL;
    AI_Pmasla_posle_GNS_newHW : LREAL;
    AI_Pmasla_posle_GNS_LW : LREAL;
    AI_Pmasla_posle_GNS_newLW : LREAL;
    AI_Pmasla_posle_NU_HL : LREAL;
    AI_Pmasla_posle_NU_LL : LREAL;
    AI_Pmasla_posle_NU_command : UINT;
    AI_Pmasla_posle_NU_newHL : LREAL;
    AI_Pmasla_posle_NU_newLL : LREAL;
    AI_Pmasla_posle_NU_status : UDINT;
    AI_Pmasla_posle_NU_value : LREAL;
    AI_Pmasla_posle_NU_LW : LREAL;
    AI_Pmasla_posle_NU_newLW : LREAL;
    AI_Pgaza_na_vhode_nagnetatelia_HL : LREAL;
    AI_Pgaza_na_vhode_nagnetatelia_LL : LREAL;
    AI_Pgaza_na_vhode_nagnetatelia_command : UINT;
    AI_Pgaza_na_vhode_nagnetatelia_newHL : LREAL;
    AI_Pgaza_na_vhode_nagnetatelia_newLL : LREAL;
    AI_Pgaza_na_vhode_nagnetatelia_status : UDINT;
    AI_Pgaza_na_vhode_nagnetatelia_value : LREAL;
    AI_Pgaza_na_vhode_nagnetatelia_LW : LREAL;
    AI_Pgaza_na_vhode_nagnetatelia_newLW : LREAL;
    AI_Pgaza_na_vyhode_nagnetatelia_HL : LREAL;
    AI_Pgaza_na_vyhode_nagnetatelia_LL : LREAL;
    AI_Pgaza_na_vyhode_nagnetatelia_command : UINT;
    AI_Pgaza_na_vyhode_nagnetatelia_newHL : LREAL;
    AI_Pgaza_na_vyhode_nagnetatelia_newLL : LREAL;
    AI_Pgaza_na_vyhode_nagnetatelia_status : UDINT;
    AI_Pgaza_na_vyhode_nagnetatelia_value : LREAL;
    AI_Pgaza_na_vyhode_nagnetatelia_LW : LREAL;
    AI_Pgaza_na_vyhode_nagnetatelia_newLW : LREAL;
    AI_Pgaza_na_vyhode_nagnetatelia_HA : LREAL;
    AI_Pgaza_na_vyhode_nagnetatelia_newHA : LREAL;
    AI_Pimpuls_gaz_HL : LREAL;
    AI_Pimpuls_gaz_LL : LREAL;
    AI_Pimpuls_gaz_command : UINT;
    AI_Pimpuls_gaz_newHL : LREAL;
    AI_Pimpuls_gaz_newLL : LREAL;
    AI_Pimpuls_gaz_status : UDINT;
    AI_Pimpuls_gaz_value : LREAL;
    AI_Pimpuls_gaz_LW : LREAL;
    AI_Pimpuls_gaz_newLW : LREAL;
    AI_dPgaza_na_maslo_filtre_HL : LREAL;
    AI_dPgaza_na_maslo_filtre_LL : LREAL;
    AI_dPgaza_na_maslo_filtre_command : UINT;
    AI_dPgaza_na_maslo_filtre_newHL : LREAL;
    AI_dPgaza_na_maslo_filtre_newLL : LREAL;
    AI_dPgaza_na_maslo_filtre_status : UDINT;
    AI_dPgaza_na_maslo_filtre_value : LREAL;
    AI_dPgaza_na_maslo_filtre_HW : LREAL;
    AI_dPgaza_na_maslo_filtre_newHW : LREAL;
    AI_dPgaza_na_konfuzore_HL : LREAL;
    AI_dPgaza_na_konfuzore_LL : LREAL;
    AI_dPgaza_na_konfuzore_command : UINT;
    AI_dPgaza_na_konfuzore_newHL : LREAL;
    AI_dPgaza_na_konfuzore_newLL : LREAL;
    AI_dPgaza_na_konfuzore_status : UDINT;
    AI_dPgaza_na_konfuzore_value : LREAL;
    AI_dPgaza_na_konfuzore_LW : LREAL;
    AI_dPgaza_na_konfuzore_newLW : LREAL;
    AI_dPmaslo_gaz_HL : LREAL;
    AI_dPmaslo_gaz_LL : LREAL;
    AI_dPmaslo_gaz_command : UINT;
    AI_dPmaslo_gaz_newHL : LREAL;
    AI_dPmaslo_gaz_newLL : LREAL;
    AI_dPmaslo_gaz_status : UDINT;
    AI_dPmaslo_gaz_value : LREAL;
    AI_dPmaslo_gaz_LW : LREAL;
    AI_dPmaslo_gaz_newLW : LREAL;
    AI_dPmaslo_gaz_LA : LREAL;
    AI_dPmaslo_gaz_newLA : LREAL;
    AI_Os_sdvig_nagnetatelja_plus_HL : LREAL;
    AI_Os_sdvig_nagnetatelja_plus_LL : LREAL;
    AI_Os_sdvig_nagnetatelja_plus_command : UINT;
    AI_Os_sdvig_nagnetatelja_plus_newHL : LREAL;
    AI_Os_sdvig_nagnetatelja_plus_newLL : LREAL;
    AI_Os_sdvig_nagnetatelja_plus_status : UDINT;
    AI_Os_sdvig_nagnetatelja_plus_value : LREAL;
    AI_Os_sdvig_nagnetatelja_plus_HW : LREAL;
    AI_Os_sdvig_nagnetatelja_plus_newHW : LREAL;
    AI_Os_sdvig_nagnetatelja_plus_HA : LREAL;
    AI_Os_sdvig_nagnetatelja_plus_newHA : LREAL;
    AI_Os_sdvig_nagnetatelja_minus_HL : LREAL;
    AI_Os_sdvig_nagnetatelja_minus_LL : LREAL;
    AI_Os_sdvig_nagnetatelja_minus_command : UINT;
    AI_Os_sdvig_nagnetatelja_minus_newHL : LREAL;
    AI_Os_sdvig_nagnetatelja_minus_newLL : LREAL;
    AI_Os_sdvig_nagnetatelja_minus_status : UDINT;
    AI_Os_sdvig_nagnetatelja_minus_value : LREAL;
    AI_Os_sdvig_nagnetatelja_minus_LW : LREAL;
    AI_Os_sdvig_nagnetatelja_minus_newLW : LREAL;
    AI_Os_sdvig_nagnetatelja_minus_LA : LREAL;
    AI_Os_sdvig_nagnetatelja_minus_newLA : LREAL;
    AI_Yroven_masla_MB_HL : LREAL;
    AI_Yroven_masla_MB_LL : LREAL;
    AI_Yroven_masla_MB_command : UINT;
    AI_Yroven_masla_MB_newHL : LREAL;
    AI_Yroven_masla_MB_newLL : LREAL;
    AI_Yroven_masla_MB_status : UDINT;
    AI_Yroven_masla_MB_value : LREAL;
    AI_Yroven_masla_MB_LW : LREAL;
    AI_Yroven_masla_MB_newLW : LREAL;
    AI_Kontrol_per_220V_HL : LREAL;
    AI_Kontrol_per_220V_LL : LREAL;
    AI_Kontrol_per_220V_command : UINT;
    AI_Kontrol_per_220V_newHL : LREAL;
    AI_Kontrol_per_220V_newLL : LREAL;
    AI_Kontrol_per_220V_status : UDINT;
    AI_Kontrol_per_220V_value : LREAL;
    AI_Kontrol_per_220V_HW : LREAL;
    AI_Kontrol_per_220V_newHW : LREAL;
    AI_Kontrol_per_220V_LW : LREAL;
    AI_Kontrol_per_220V_newLW : LREAL;
    AI_Kontrol_post_220V_HL : LREAL;
    AI_Kontrol_post_220V_LL : LREAL;
    AI_Kontrol_post_220V_command : UINT;
    AI_Kontrol_post_220V_newHL : LREAL;
    AI_Kontrol_post_220V_newLL : LREAL;
    AI_Kontrol_post_220V_status : UDINT;
    AI_Kontrol_post_220V_value : LREAL;
    AI_Kontrol_post_220V_HW : LREAL;
    AI_Kontrol_post_220V_newHW : LREAL;
    AI_Kontrol_post_220V_LW : LREAL;
    AI_Kontrol_post_220V_newLW : LREAL;
    AI_Tok_statora_HL : LREAL;
    AI_Tok_statora_LL : LREAL;
    AI_Tok_statora_command : UINT;
    AI_Tok_statora_newHL : LREAL;
    AI_Tok_statora_newLL : LREAL;
    AI_Tok_statora_status : UDINT;
    AI_Tok_statora_value : LREAL;
    AI_Tok_statora_LW : LREAL;
    AI_Tok_statora_newLW : LREAL;
    AI_Vibro_skorost_OPED_T1_HL : LREAL;
    AI_Vibro_skorost_OPED_T1_LL : LREAL;
    AI_Vibro_skorost_OPED_T1_command : UINT;
    AI_Vibro_skorost_OPED_T1_newHL : LREAL;
    AI_Vibro_skorost_OPED_T1_newLL : LREAL;
    AI_Vibro_skorost_OPED_T1_status : UDINT;
    AI_Vibro_skorost_OPED_T1_value : LREAL;
    AI_Vibro_skorost_OPED_T1_HW : LREAL;
    AI_Vibro_skorost_OPED_T1_newHW : LREAL;
    AI_Vibro_skorost_OPED_T1_HA : LREAL;
    AI_Vibro_skorost_OPED_T1_newHA : LREAL;
    AI_Vibro_skorost_OYPED_T2_HL : LREAL;
    AI_Vibro_skorost_OYPED_T2_LL : LREAL;
    AI_Vibro_skorost_OYPED_T2_command : UINT;
    AI_Vibro_skorost_OYPED_T2_newHL : LREAL;
    AI_Vibro_skorost_OYPED_T2_newLL : LREAL;
    AI_Vibro_skorost_OYPED_T2_status : UDINT;
    AI_Vibro_skorost_OYPED_T2_value : LREAL;
    AI_Vibro_skorost_OYPED_T2_HW : LREAL;
    AI_Vibro_skorost_OYPED_T2_newHW : LREAL;
    AI_Vibro_skorost_OYPED_T2_HA : LREAL;
    AI_Vibro_skorost_OYPED_T2_newHA : LREAL;
    AI_Vibro_skorost_OYP_kolesa_ED_T3_HL : LREAL;
    AI_Vibro_skorost_OYP_kolesa_ED_T3_LL : LREAL;
    AI_Vibro_skorost_OYP_kolesa_ED_T3_command : UINT;
    AI_Vibro_skorost_OYP_kolesa_ED_T3_newHL : LREAL;
    AI_Vibro_skorost_OYP_kolesa_ED_T3_newLL : LREAL;
    AI_Vibro_skorost_OYP_kolesa_ED_T3_status : UDINT;
    AI_Vibro_skorost_OYP_kolesa_ED_T3_value : LREAL;
    AI_Vibro_skorost_OYP_kolesa_ED_T3_HW : LREAL;
    AI_Vibro_skorost_OYP_kolesa_ED_T3_newHW : LREAL;
    AI_Vibro_skorost_OYP_kolesa_ED_T3_HA : LREAL;
    AI_Vibro_skorost_OYP_kolesa_ED_T3_newHA : LREAL;
    AI_Vibro_skorost_OP_kolesa_RH_T4_HL : LREAL;
    AI_Vibro_skorost_OP_kolesa_RH_T4_LL : LREAL;
    AI_Vibro_skorost_OP_kolesa_RH_T4_command : UINT;
    AI_Vibro_skorost_OP_kolesa_RH_T4_newHL : LREAL;
    AI_Vibro_skorost_OP_kolesa_RH_T4_newLL : LREAL;
    AI_Vibro_skorost_OP_kolesa_RH_T4_status : UDINT;
    AI_Vibro_skorost_OP_kolesa_RH_T4_value : LREAL;
    AI_Vibro_skorost_OP_kolesa_RH_T4_HW : LREAL;
    AI_Vibro_skorost_OP_kolesa_RH_T4_newHW : LREAL;
    AI_Vibro_skorost_OP_kolesa_RH_T4_HA : LREAL;
    AI_Vibro_skorost_OP_kolesa_RH_T4_newHA : LREAL;
    AI_Vibro_skorost_OP_shesterni_RED_T5_HL : LREAL;
    AI_Vibro_skorost_OP_shesterni_RED_T5_LL : LREAL;
    AI_Vibro_skorost_OP_shesterni_RED_T5_command : UINT;
    AI_Vibro_skorost_OP_shesterni_RED_T5_newHL : LREAL;
    AI_Vibro_skorost_OP_shesterni_RED_T5_newLL : LREAL;
    AI_Vibro_skorost_OP_shesterni_RED_T5_status : UDINT;
    AI_Vibro_skorost_OP_shesterni_RED_T5_value : LREAL;
    AI_Vibro_skorost_OP_shesterni_RED_T5_HW : LREAL;
    AI_Vibro_skorost_OP_shesterni_RED_T5_newHW : LREAL;
    AI_Vibro_skorost_OP_shesterni_RED_T5_HA : LREAL;
    AI_Vibro_skorost_OP_shesterni_RED_T5_newHA : LREAL;
    AI_Vibro_skorost_OP_shesterni_RED_T6_HL : LREAL;
    AI_Vibro_skorost_OP_shesterni_RED_T6_LL : LREAL;
    AI_Vibro_skorost_OP_shesterni_RED_T6_command : UINT;
    AI_Vibro_skorost_OP_shesterni_RED_T6_newHL : LREAL;
    AI_Vibro_skorost_OP_shesterni_RED_T6_newLL : LREAL;
    AI_Vibro_skorost_OP_shesterni_RED_T6_status : UDINT;
    AI_Vibro_skorost_OP_shesterni_RED_T6_value : LREAL;
    AI_Vibro_skorost_OP_shesterni_RED_T6_HW : LREAL;
    AI_Vibro_skorost_OP_shesterni_RED_T6_newHW : LREAL;
    AI_Vibro_skorost_OP_shesterni_RED_T6_HA : LREAL;
    AI_Vibro_skorost_OP_shesterni_RED_T6_newHA : LREAL;
  END_VAR
